(* IEC 61131-3 sources: MotionTestBenchMaster/Logical/00_AID/Libraries/Sidel_Libraries/Sidel_Obj, 21 files *)

(* ---- HMI_Structure.typ ---- *)
(*VALVES*)

TYPE
	HMI_Valve_Type : 	STRUCT  (*Valves Structure: Digital*)
		Out : BOOL; (*State: Output*)
		Alarm : BOOL; (*State: Position Alarm *)
		Opened : BOOL; (*State: Feed-Back Opened*)
		Closed : BOOL; (*State: Feed-Back Closed*)
		ConfigPosition : BOOL; (*Configuration: Valve Feed-Back Position Present *)
		ConfigPresent : BOOL; (*Configuration: Device Present*)
		ManOff : BOOL; (*Command: Manual Closed*)
		ManOn : BOOL; (*Command: Manual Opened *)
		Mask : BOOL; (*Command: Position Alarm Mask*)
		ManEnable : BOOL; (*Command Enable: Manual Enabled*)
		MaskEnable : BOOL; (*Command Enable: Mask Enabled*)
	END_STRUCT;
	HMI_Valve_MixProof_Type : 	STRUCT  (*Valves Structure: Digital Mix Proof*)
		Out : BOOL; (*State: Output*)
		Alarm : BOOL; (*State: Position Alarm *)
		Opened : BOOL; (*State: Feed-Back Opened*)
		Closed : BOOL; (*State: Feed-Back Closed*)
		ConfigPosition : BOOL; (*Configuration: Valve Feed-Back Position Present *)
		ConfigPresent : BOOL; (*Configuration: Device Present*)
		ManOff : BOOL; (*Command: Manual Closed*)
		ManOn : BOOL; (*Command: Manual Opened *)
		Mask : BOOL; (*Command: Position Alarm Mask*)
		ManEnable : BOOL; (*Command Enable: Manual Enabled*)
		MaskEnable : BOOL; (*Command Enable: Mask Enabled*)
		H_Out : BOOL; (*High State: Output*)
		H_Alarm : BOOL; (*High State: Position Alarm *)
		H_Opened : BOOL; (*High State: Feed-Back Opened*)
		H_Closed : BOOL; (*High State: Feed-Back Closed*)
		H_ConfigPosition : BOOL; (*High Configuration: Valve Closed State Present *)
		H_ManOff : BOOL; (*High Command: Manual Closed*)
		H_ManOn : BOOL; (*High Command: Manual Opened *)
		H_Mask : BOOL; (*High Command: Position Alarm Mask*)
		H_ManEnable : BOOL; (*High Command Enable: Manual Enabled*)
		H_MaskEnable : BOOL; (*High Command Enable: Mask Enabled*)
		L_Out : BOOL; (*Low State: Output*)
		L_Alarm : BOOL; (*Low State: Position Alarm *)
		L_Opened : BOOL; (*Low State: Feed-Back Opened*)
		L_Closed : BOOL; (*Low State: Feed-Back Closed*)
		L_ConfigPosition : BOOL; (*Low Configuration: Valve Closed State Present *)
		L_ManOff : BOOL; (*Low Command: Manual Closed*)
		L_ManOn : BOOL; (*Low Command: Manual Opened *)
		L_Mask : BOOL; (*Low Command: Position Alarm Mask*)
		L_ManEnable : BOOL; (*Low Command Enable: Manual Enabled*)
		L_MaskEnable : BOOL; (*Low Command Enable: Mask Enabled*)
	END_STRUCT;
	HMI_Valve_Mod_Type : 	STRUCT  (*Valves Structure: Analogic*)
		Out : BOOL; (*State: Output*)
		Alarm : BOOL; (*State: Position Alarm *)
		Opened : BOOL; (*State: Feed-Back Opened*)
		Closed : BOOL; (*State: Feed-Back Closed*)
		ConfigSlew : BOOL; (*Configuration: Output Slew Present*)
		ConfigPosition : BOOL; (*Configuration: Valve Feed-Back Position Present *)
		ConfigPresent : BOOL; (*Configuration: Device Present*)
		ManOff : BOOL; (*Command: Manual Closed*)
		ManOn : BOOL; (*Command: Drive Manual OUT = OUT_Man*)
		Mask : BOOL; (*Command: Position Alarm Mask*)
		ManEnable : BOOL; (*Command Enable: Manual Enabled*)
		MaskEnable : BOOL; (*Command Enable: Mask Enabled*)
		OUT_CV : REAL; (*State: Actual OUTPUT Control Value (0.0-:-100.0)*)
		OUT_Man : REAL; (*Command: Manual OUTPUT Value (0.0-:-100.0)*)
		FBK : REAL; (*State: Feed-Back INPUT Value (0.0-:-100.0)*)
	END_STRUCT;
END_TYPE

(*MOTORS*)

TYPE
	HMI_SCU_Type : 	STRUCT
		Visibility : BOOL;
		Alarm : BOOL;
		ErrCode : DINT;
		HwCmdUp : BOOL;
		HwCmdDown : BOOL;
		HwCmdStorePosition : BOOL;
	END_STRUCT;
	HMI_Column_Type : 	STRUCT
		Visibility : BOOL;
		Running : BOOL; (*State: Output*)
		Current : REAL;
		Initialized : BOOL;
		Position : REAL;
		Alarm : BOOL;
	END_STRUCT;
	HMI_Motor_Type : 	STRUCT  (*Motor Structure: Direct On Line*)
		Out : BOOL; (*State: Running*)
		Alarm : BOOL; (*State: Alarm (Isolated, Overload, FBK Fault)*)
		Isolated : BOOL; (*State: Motor Isolated*)
		Overload : BOOL; (*State: Overload*)
		FeedBack : BOOL; (*State: Feed-Back Fault*)
		ConfigPresent : BOOL; (*Configuration: Device Present*)
		ManOff : BOOL; (*Command: Manual Stop*)
		ManOn : BOOL; (*Command: Manual Start*)
		Mask : BOOL; (*Command: Alarm Mask*)
		ManEnable : BOOL; (*Command Enable: Manual Enabled*)
		MaskEnable : BOOL; (*Command Enable: Mask Enabled*)
	END_STRUCT;
	HMI_Motor_FC_Type : 	STRUCT  (*Motor Structure: Variable Frequency Drive*)
		Out : BOOL; (*State: Running *)
		Alarm : BOOL; (*State: Alarm (Isolated, Overload, FBK Fault)*)
		Isolated : BOOL; (*State: Motor Isolated*)
		Overload : BOOL; (*State: Overload*)
		FeedBack : BOOL; (*State: In Operation/Safe-OFF Feed-Back Fault*)
		BusFault : BOOL; (*State: Bus Control Fault*)
		Fault : BOOL; (*State: Inverter Internal Fault*)
		ConfigPresent : BOOL; (*Configuration: Device Present*)
		ManOff : BOOL; (*Command: Manual Stop*)
		ManOn : BOOL; (*Command: Manual Start*)
		Mask : BOOL; (*Command: Alarm Mask*)
		ManEnable : BOOL; (*Command Enable: Manual Enabled*)
		MaskEnable : BOOL; (*Command Enable: Mask Enabled*)
		OUT_CV : REAL; (*State: Actual OUTPUT Value (0.0-:-100.0)*)
		OUT_Man : REAL; (*Command: Manual OUTPUT Value (0.0-:-100.0)*)
	END_STRUCT;
	HMI_Dosing_Pump_Type : 	STRUCT  (*Motor Structure: Dosing Pump*)
		Out : BOOL; (*State: Running *)
		Alarm : BOOL; (*State: Alarm (Isolated, Overload, FBK Fault)*)
		Isolated : BOOL; (*State: Motor Isolated*)
		Overload : BOOL; (*State: Overload*)
		FeedBack : BOOL; (*State: In Operation/Safe-OFF Feed-Back Fault*)
		Pulse_FBK : BOOL; (*State: Pulse Feed-Back Alarm*)
		Internal_Fault : BOOL; (*State: Internal Alarm*)
		ConfigPresent : BOOL; (*Configuration: Device Present*)
		ManOff : BOOL; (*Command: Manual Stop*)
		ManOn : BOOL; (*Command: Manual Start *)
		Mask : BOOL; (*Command: Alarm Mask*)
		ManEnable : BOOL; (*Command Enable: Manual Enabled*)
		MaskEnable : BOOL; (*Command Enable: Mask Enabled*)
		Stroke_Value : REAL; (*Setting CC/Stroke [cm3/stroke]*)
		Concentration : REAL; (*Tank Concentrated percentage [0..1000000 ppm]*)
		Density : REAL; (*Specific Weight [kg]*)
	END_STRUCT;
	HMI_Danfoss_Diag_Type : 	STRUCT
		PCV : HMI_Danfoss_PCV_Type;
		PCD_Read : HMI_Danfoss_PCD_Read_Type;
	END_STRUCT;
	HMI_Danfoss_PCV_Type : 	STRUCT
		Alarm : DINT;
	END_STRUCT;
	HMI_Danfoss_PCD_Read_Type : 	STRUCT
		Power : REAL;
		Motor_Current : REAL;
		Frequency : REAL;
		Torque : REAL;
		Main_Actual_Value : REAL;
		Speed_RPM : REAL;
		Status_Word : UINT;
	END_STRUCT;
	HMI_Fan_Type : 	STRUCT
		HMI_Pressurizer : ARRAY[1..6]OF HMI_Pressurizer_Type; (*Single Fans to HMI*)
		HMI_Galvani : HMI_Galvani_Type; (*Galvani Roof Fans*)
	END_STRUCT;
	HMI_Galvani_Type : 	STRUCT
		Out : BOOL;
		ConfigPresent : BOOL; (*Configuration: Device Present*)
		SS2P_Lamp1 : HMI_SS2P_Type; (*SS2P Lamp*)
		SS2P_Lamp2 : HMI_SS2P_Type; (*SS2P Lamp*)
		ManState : BOOL; (*State: Device in manual mode*)
		ManEnable : BOOL; (*Command Enable: Manual Enabled*)
		ManFlowSet : BOOL; (*Command: Manual Flow set command*)
		ManOff : BOOL; (*Command: Manual Stop*)
		ManOn : BOOL; (*Command: Manual Start*)
		MaskEnable : BOOL; (*Command Enable: Mask Enabled*)
		Mask : BOOL; (*Command: Alarm Mask*)
		FlowSet : BOOL; (*State: Flow set speed *)
		Alarm : BOOL; (*State: Alarm (Isolated, Overload, FBK Fault)*)
		AlarmAbsoluteFilter : BOOL; (*Fault : Absolute filter clogged*)
		AlarmPrefilterExt : BOOL; (*Fault : External PreFilter Clogged*)
		AlarmPrefilterInt : BOOL; (*Fault : Internal PreFilter Clogged*)
		Overload : BOOL; (*State: Power supply on*)
	END_STRUCT;
	HMI_Pressurizer_Type : 	STRUCT
		Out : BOOL;
		ConfigPresent : BOOL; (*Configuration: Device Present*)
		SS2P_Lamp : HMI_SS2P_Type; (*SS2P Lamp*)
		ManState : BOOL; (*State: Device in manual mode*)
		ManEnable : BOOL; (*Command Enable: Manual Enabled*)
		ManOff : BOOL; (*Command: Manual Stop*)
		ManOn : BOOL; (*Command: Manual Start*)
		MaskEnable : BOOL; (*Command Enable: Mask Enabled*)
		Mask : BOOL; (*Command: Alarm Mask*)
		OUT_Man : REAL; (*Command :  Manual Speed OUT value selected (0 - 100)*)
		OUT_CV : REAL; (*State : Actual Speed OUT value %*)
		Alarm : BOOL; (*State: Alarm (Isolated, Overload, FBK Fault)*)
		AlarmFilter : BOOL; (*Fault : Absolute filter or PreFilter Clogged*)
	END_STRUCT;
	HMI_GreasingPump_Type : 	STRUCT
		LowLevel : HMI_DI_Type;
		CycleEnd : HMI_DI_Type;
		Motor : HMI_Motor_Type;
	END_STRUCT;
END_TYPE

(*INSTRUMENTS*)

TYPE
	HMI_Valve_Ejector_Type : 	STRUCT  (*Valves Structure: Digital*)
		Out : BOOL; (*State: Output*)
		Alarm : BOOL; (*State: Position Alarm *)
		Opened : BOOL; (*State: Feed-Back Opened*)
		Closed : BOOL; (*State: Feed-Back Closed*)
		ConfigPosition : BOOL; (*Configuration: Valve Feed-Back Position Present *)
		ConfigPresent : BOOL; (*Configuration: Device Present*)
		ManOff : BOOL; (*Command: Manual Closed*)
		ManOn : BOOL; (*Command: Manual Opened *)
		Mask : BOOL; (*Command: Position Alarm Mask*)
		ManEnable : BOOL; (*Command Enable: Manual Enabled*)
		MaskEnable : BOOL; (*Command Enable: Mask Enabled*)
		CounterReset : BOOL; (*Command: Reset Counter*)
		TotalErrors : UDINT; (*State : Total Errors*)
		AbsoluteErrors : USINT; (*State : Absolute Errors*)
		ConsecutiveErrors : USINT; (*State : Consecutive Errors*)
	END_STRUCT;
	HMI_Photocell_Type : 	STRUCT  (*Instrument Structure: Photocell*)
		On : BOOL; (*State: Active*)
		Alarm : BOOL; (*State: Alarm*)
		Wait : BOOL; (*State: Waiting condition*)
		ConfigAlarm : BOOL; (*Configuration: Alarm Present*)
		ConfigPresent : BOOL; (*Configuration: Instrument Present*)
		Mask : BOOL; (*Command: Alarm Mask*)
		MaskEnable : BOOL; (*Command Enable: Mask Enabled*)
		CounterReset : BOOL; (*Command: Reset Counter*)
		TotalErrors : UDINT; (*State : Total Errors*)
		RepetitiveErrors : USINT; (*State : Repetitive Errors*)
		AbsoluteErrors : USINT; (*State : Absolute Errors*)
		ConsecutiveErrors : USINT; (*State : Consecutive Errors*)
		AlwaysTrueSteps : USINT;
	END_STRUCT;
	HMI_DI_Type : 	STRUCT  (*Instrument Structure: Digital*)
		On : BOOL; (*State: Active*)
		Alarm : BOOL; (*State: Alarm*)
		Wait : BOOL; (*State: Waiting condition*)
		ConfigAlarm : BOOL; (*Configuration: Alarm Present*)
		ConfigPresent : BOOL; (*Configuration: Instrument Present*)
		Mask : BOOL; (*Command: Alarm Mask*)
		MaskEnable : BOOL; (*Command Enable: Mask Enabled*)
	END_STRUCT;
	HMI_Analog_IN_Type : 	STRUCT  (*Instrument Structure: Analogic*)
		Alarm : BOOL; (*State: Instrument in fault (Probe Fault)*)
		Wait : BOOL; (*State: Waiting condition*)
		WaitCounter : BOOL; (*State: Waiting Counter condition*)
		ConfigPopUp : BOOL; (*Configuration: Instrument Pop-Up Present (TRUE=Pop-Up NOT Present)*)
		ConfigTot : BOOL; (*Configuration: Totalizator Present (TRUE=Totalizator Present)*)
		ConfigAlarm : BOOL; (*Configuration: Alarm Present (TRUE=Command Mask Present)*)
		ConfigPresent : BOOL; (*Configuration: Instrument Present*)
		ConfigCounter : BOOL; (*Configuration: Counter Present*)
		ResetTot : BOOL; (*Command: Totalizator Reset*)
		Mask : BOOL; (*Command: Alarm Mask (Probe Fault disabled)*)
		MaskEnable : BOOL; (*Command Enable: Mask Enabled*)
		PV : REAL; (*Input: Scaled Process Value*)
		SP : REAL; (*Input: Actual SetPoint*)
		PV_Counter : REAL; (*Input: Counter Current Value*)
		SP_Counter : REAL; (*Input: Counter Requested Value*)
		Tot : REAL; (*Input: Totalizator*)
	END_STRUCT;
	HMI_Analog_IN_Mode_Type : 	STRUCT  (*Instrument Structure: Analogic Multi Scale*)
		Mode : ARRAY[0..3]OF HMI_Analog_IN_Type;
	END_STRUCT;
	HMI_Analog_Multiscale_Type : 	STRUCT  (*Instrument Structure: Analogic*)
		Alarm : BOOL; (*State: Instrument in fault (Probe Fault)*)
		Unit : USINT; (*0 = Unit1 ; 1 = Unit2 ; 2 = Unit3 ; etc...*)
		ConfigPopup : BOOL; (*Configuration: Instrument Pop-Up Present (TRUE=Pop-Up NOT Present)*)
		ConfigAlarm : BOOL; (*Configuration: Alarm Present (TRUE=Command Mask Present)*)
		ConfigPresent : BOOL; (*Configuration: Instrument Present*)
		ResetTot : BOOL; (*Command: Totalizator Reset*)
		Mask : BOOL; (*Command: Alarm Mask (Probe Fault disabled)*)
		MaskEnable : BOOL; (*Command Enable: Mask Enabled*)
		Wait : ARRAY[0..3]OF BOOL; (*State: Waiting condition*)
		ConfigTot : ARRAY[0..3]OF BOOL; (*Configuration: Totalizator Present (TRUE=Totalizator Present)*)
		WaitCounter : ARRAY[0..3]OF BOOL; (*State: Waiting Counter condition*)
		ConfigCounter : ARRAY[0..3]OF BOOL; (*Configuration: Counter Present*)
		PV : ARRAY[0..3]OF REAL; (*Input: Scaled Process Value*)
		SP : ARRAY[0..3]OF REAL; (*Input: Actual SetPoint*)
		PV_Counter : ARRAY[0..3]OF REAL; (*Input: Counter Current Value*)
		SP_Counter : ARRAY[0..3]OF REAL; (*Input: Counter Requested Value*)
		Tot : ARRAY[0..3]OF REAL; (*Input: Totalizator*)
	END_STRUCT;
	HMI_TNK_Level_Type : 	STRUCT
		CFG_Level_Percentage : BOOL;
		Level_Percentage : REAL; (*[%]*)
		CFG_Level_Percentage_SP : BOOL; (*[%]*)
		Level_Height_SP : REAL; (*[mm]*)
		Level_Percentage_SP : REAL; (*[%]*)
		CFG_Volume : BOOL;
		Volume : REAL; (*[l]*)
		CFG_Volume_SP : BOOL; (*[l]*)
		Level_Percentage_Wait : BOOL;
		Level_Height_Wait : BOOL;
		Volume_Wait : BOOL;
		Volume_SP : REAL; (*[l]*)
		CFG_Level_Height : BOOL;
		Level_Height : REAL; (*[mm]*)
	END_STRUCT;
	HMI_TNK_Level_v00_Type : 	STRUCT
		ConfigPresent : BOOL := TRUE;
		TNK_Height_mm : REAL; (*[mm]*)
		TNK_Height_Sp : REAL; (*[mm]*)
		TNK_Height_Wait : BOOL;
		TNK_Percentage : REAL; (*[%]*)
		TNK_Percentage_Sp : REAL; (*[%]*)
		TNK_Percentage_Wait : BOOL;
		TNK_Volume_liters : REAL; (*[l]*)
		TNK_Volume_Sp : REAL; (*[l]*)
		TNK_Volume_Wait : BOOL;
	END_STRUCT;
	HMI_GateDoor_Type : 	STRUCT
		Opened : BOOL;
		ShortSafety : BOOL;
		Production : HMI_DI_Type;
		Cleaning : HMI_DI_Type;
	END_STRUCT;
END_TYPE

(*PID*)

TYPE
	HMI_PID_Mode_Type : 	STRUCT
		Mode : ARRAY[0..3]OF HMI_PID_Type;
	END_STRUCT;
	HMI_PID_Type : 	STRUCT  (*PID Structure: PID Control*)
		Enable : BOOL; (*State: PID Enable*)
		Mode : BOOL; (*State: PID Mode (Automatic = 1  Manual = 0)*)
		Alarm : BOOL; (*State: PID PV in fault*)
		SP_Obtained : BOOL; (*State: PID Set Point Reached*)
		SP_SlewRunning : BOOL; (*State: PID Set Point Slew Running*)
		CnScale : BOOL; (*Configuration: FF and PID OUT Scale - TRUE-> 0-100%, FALSE-> Ing.Unit.*)
		ConfigSlewPresent : BOOL; (*Configuration: Slew Present*)
		ConfigPresent : BOOL; (*Configuration : PID present*)
		SPLocal : BOOL; (*Command: PID Manual Set Point -> "SP_Local"*)
		PV : REAL; (*State: PID Process Value*)
		SP_Actual : REAL; (*State: PID Set Point in Use*)
		SP_Target : REAL; (*State: PID Set Point*)
		FF_OUT : REAL; (*State: PID Feed Forward calculated value*)
		OUT : REAL; (*State: PID Output*)
		SP_Local : REAL; (*Command: PID Manual Set Point Target Value*)
	END_STRUCT;
END_TYPE

(*PWM*)

TYPE
	HMI_PWM_Type : 	STRUCT  (*PWM Structure: Pulse Width Modulation*)
		Out : BOOL; (*State: On*)
		Alarm : BOOL; (*State: Alarm (Isolated, Overload, FBK Fault)*)
		Isolated : BOOL; (*State: Isolated*)
		Overload : BOOL; (*State: Overload*)
		FeedBack : BOOL; (*State: Feed-Back Fault*)
		ConfigPresent : BOOL; (*Configuration: Device Present*)
		ManOff : BOOL; (*Command: Manual Stop*)
		ManOn : BOOL; (*Command: Manual Start*)
		Mask : BOOL; (*Command: Alarm Mask*)
		ManEnable : BOOL; (*Command Enable: Manual Enabled*)
		MaskEnable : BOOL; (*Command Enable: Mask Enabled*)
		OUT_CV : REAL; (*State: Actual OUTPUT Control Value (0.0-:-100.0)*)
		OUT_Man : REAL; (*Command: Manual OUTPUT Value (0.0-:-100.0)*)
	END_STRUCT;
END_TYPE

(* *)

TYPE
	HMI_SS2P_Type : 	STRUCT  (*Selector 2 position (Auto-Man; ON-OFF;) 0=Auto/OFF - 1=Man/ON*)
		Enable : BOOL; (*State: Command Enabled*)
		LampON : BOOL; (*State: Lamp Command ON*)
		Blink : BOOL; (*State: Blink LampOn*)
		Visibility : BOOL; (*Configuration: Present*)
		ON : BOOL; (*Command: Selector Button ON*)
	END_STRUCT;
END_TYPE

(* ---- IO_Structure.typ ---- *)
(*VALVES*)

TYPE
	IO_Valve_Mod_Type : 	STRUCT
		AO_Raw : INT;
		AI_Raw : INT;
		Valve : IO_Valve_Type;
	END_STRUCT;
	IO_ValveMac_Type : 	STRUCT
		DI_PowerSupplyPhyChannelOk : BOOL;
		DI_Opened : BOOL; (*DI Valve Open - Feedback*)
		DI_Closed : BOOL; (*DI Valve Close - Feedback*)
		DO_Opened : BOOL; (*DO Valve Open*)
		DO_Closed : BOOL; (*DO Valve Close*)
	END_STRUCT;
	IO_Valve_Type : 	STRUCT
		DI_Opened : BOOL; (*DI Valve Open - Feedback*)
		DI_Closed : BOOL; (*DI Valve Close - Feedback*)
		DO_Opened : BOOL; (*DO Valve Open*)
		DO_Closed : BOOL; (*DO Valve Close*)
	END_STRUCT;
END_TYPE

(*MOTORS*)

TYPE
	IO_Motor_FwBw_Type : 	STRUCT  (*Motor control Forward Backward*)
		DI_SafetyEnable : BOOL; (*Safety Enable from IOMapping*)
		DI_SafetyFault : BOOL; (*Safety Feed-Back from Safety CPU*)
		DI_Fault : BOOL;
		DI_ContactorFBK : BOOL; (*Contactor Feed-Back *)
		DI_OverloadOK : BOOL := TRUE; (*Not present in case of UL*)
		DI_ManSwitchON : BOOL := TRUE;
		DO_MotorFw : BOOL; (*Start Forward*)
		DO_MotorBw : BOOL; (*Start Backward*)
	END_STRUCT;
	IO_MotorFC280_Type : 	STRUCT  (*Motor control*)
		DI_SafetyEnable : BOOL; (*Safety Enable from IOMapping*)
		DI_SafetyFault : BOOL; (*Safety Feed-Back from Safety CPU*)
		DI_ManSwitchON : BOOL := TRUE;
		DI_ContactorFBK : BOOL; (*Contactor Feed-Back *)
		DI_OverloadOK : BOOL := TRUE; (*Not present in case of UL*)
		DO_MotorON : BOOL; (*Start*)
		DO_ShuntTrip : BOOL; (*Thermal Protection Forced Trip*)
	END_STRUCT;
	IO_Motor_Type : 	STRUCT  (*Motor control*)
		DI_SafetyEnable : BOOL; (*Safety Enable from IOMapping*)
		DI_SafetyFault : BOOL; (*Safety Feed-Back from Safety CPU*)
		DI_ManSwitchON : BOOL := TRUE;
		DI_ContactorFBK : BOOL; (*Contactor Feed-Back *)
		DI_OverloadOK : BOOL := TRUE; (*Not present in case of UL*)
		DO_MotorON : BOOL; (*Start*)
		DO_ShuntTrip : BOOL; (*Thermal Protection Forced Trip*)
	END_STRUCT;
	IO_UVtronic_Type : 	STRUCT  (*Henovia UV control*)
		DI_SafetyEnable : BOOL; (*Safety Enable from IOMapping*)
		DI_Ready : BOOL;
		DI_Alarm : BOOL;
		DI_GeneralFault : BOOL;
		DI_ContactorFBK : BOOL; (*Contactor Feed-Back *)
		DI_OverloadOK : BOOL := TRUE; (*Not present in case of UL*)
		DO_MotorON : BOOL; (*Start*)
	END_STRUCT;
	IO_PLK_DanfossFC280_Drive_Type : 	STRUCT  (*Powerlink Danfoss VLT Interface*)
		Input : IO_PLK_DanfossFC280_IN;
		Output : IO_PLK_DanfossFC280_OUT;
	END_STRUCT;
	IO_PLK_Danfoss_Drive_Type : 	STRUCT  (*Powerlink Danfoss VLT Interface*)
		Input : IO_PLK_Danfoss_IN;
		Output : IO_PLK_Danfoss_OUT;
	END_STRUCT;
	IO_PLK_DanfossFC280_IN : 	STRUCT  (*Powerlink Danfoss VLT Inputs*)
		STW : UINT; (*Status Word*)
		MAV : INT; (*Main Actual Value*)
		ActFreq : UDINT; (*Actual Frequency [Hz]*)
		ActCurrent : UINT; (*Actual Current [A]*)
		Power : UDINT; (*Power [kW]*)
		Torque : DINT; (*Torque [Nm]*)
		SpeedRPM : DINT; (*Speed [RPM]*)
		STW_EX : UDINT; (*Extended Status Word 1*)
		ErrorCode : UDINT; (*Error Code 1*)
		DigitalInput : UINT; (*Digital Input V4.A.A.1.6.13*)
	END_STRUCT;
	IO_PLK_Danfoss_IN : 	STRUCT  (*Powerlink Danfoss VLT Inputs*)
		STW : UINT; (*Status Word*)
		MAV : INT; (*Main Actual Value*)
		ActFreq : UINT; (*Actual Frequency [Hz]*)
		ActCurrent : DINT; (*Actual Current [A]*)
		Power : DINT; (*Power [kW]*)
		Torque : INT; (*Torque [Nm]*)
		SpeedRPM : DINT; (*Speed [RPM]*)
		STW_EX : UDINT; (*Extended Status Word 1*)
		ErrorCode : UDINT; (*Error Code 1*)
		DigitalInput : UINT; (*Digital Input V4.A.A.1.6.13*)
	END_STRUCT;
	IO_PLK_DanfossFC280_OUT : 	STRUCT  (*Powerlink Danfoss VLT Outputs*)
		CTW : UINT; (*Control Word*)
		MRW : INT; (*Main Reference Value*)
	END_STRUCT;
	IO_PLK_Danfoss_OUT : 	STRUCT  (*Powerlink Danfoss VLT Outputs*)
		CTW : UINT; (*Control Word*)
		MRW : INT; (*Main Reference Value*)
	END_STRUCT;
	IO_FanMain_Type : 	STRUCT
		DI_OverloadOK : BOOL := TRUE;
		DO_ZoneLighting : BOOL; (*V4.A.A.1.7.0*)
		Pressurizer : ARRAY[1..6]OF IO_Pressurizer_Type;
		GalvaniRoof : IO_GalvaniRoof_Type;
	END_STRUCT;
	IO_PressurizerMain_Type : 	STRUCT
		DI_OverloadOK : BOOL := TRUE;
		Pressurizer : ARRAY[1..6]OF IO_Pressurizer_Type;
	END_STRUCT;
	IO_GalvaniRoof_Type : 	STRUCT
		DI_Running : BOOL;
		DI_AbsoluteFilterAlarm : BOOL;
		DI_PrefilterExtAlarm : BOOL;
		DI_PrefilterIntAlarm : BOOL;
		DI_CabinetPoweredOn : BOOL;
		DO_Start : BOOL;
		DO_FlowSet : BOOL;
		DO_LightingArea_1 : BOOL;
		DO_LightingArea_2 : BOOL;
	END_STRUCT;
	IO_Pressurizer_Type : 	STRUCT
		DO_Lighting : BOOL;
		AO_Raw : INT;
		DI_PressurizerON : BOOL; (*Pressurizzer ON*)
		DI_PrefilterAlarm : BOOL; (*Pressurizzer prefilter clogged*)
		DI_AbsoluteFilterAlarm : BOOL; (*Pressurizzer absolute filter clogged*)
	END_STRUCT;
	IO_MotionFan_Type : 	STRUCT
		DI_ManSwitchON : BOOL := TRUE;
		DI_OverloadOK : BOOL := TRUE;
		DI_ContactorFBK : BOOL := TRUE;
		DO_MotorON : BOOL;
	END_STRUCT;
END_TYPE

(*INSTRUMENTS*)

TYPE
	IO_Analog_IN_OUT_Type : 	STRUCT
		AO_Raw : INT := 0; (*Analog Input From HW*)
		AI : IO_Analog_IN_Type; (*Analog Input From HW*)
	END_STRUCT;
	IO_Analog_IN_Type : 	STRUCT
		AI_Raw : INT := 0; (*Analog Input From HW*)
		DI_ChannelOk : BOOL := TRUE;
		DI_Pulse : BOOL; (*Totalizer Pulse*)
		DI_Alarm : BOOL; (*Instrument Alarm*)
		DO_SetScale : BOOL; (*Scale Change Output*)
	END_STRUCT;
	IO_Digital_IN_Type : 	STRUCT
		DI_Input : BOOL;
	END_STRUCT;
	IO_Digital_OUT_Type : 	STRUCT
		DO_Output : BOOL;
	END_STRUCT;
	IO_GreasingPump_Type : 	STRUCT
		LowLevel : IO_Digital_IN_Type;
		CycleEnd : IO_Digital_IN_Type;
		Motor : IO_Motor_Type;
	END_STRUCT;
	IN_Analog_Multiscale : 	STRUCT
		ScaleLOW : REAL;
		ScaleHIGH : REAL;
		ActualSP : REAL; (*Signal Input Actual Set Point*)
		MinDev : REAL; (*To Set Point Low Deviation (for SP obtained)*)
		MaxDev : REAL; (*To Set Point High Deviation (for SP obtained)*)
		WaitDelay : TIME;
		HighLimitEn : BOOL;
		HighLimitSP : REAL;
		HighLimitHyst : REAL;
		HighLimitDelay : TIME;
		LowLimitEn : BOOL;
		LowLimitSP : REAL;
		LowLimitHyst : REAL;
		LowLimitDelay : TIME;
		TotPulseWeight : REAL;
		TotType : USINT;
		PLCCounterSP : REAL;
		PLCCounterReset : BOOL;
		HMITotEn : BOOL;
		HMITotReset : BOOL;
	END_STRUCT;
	OUT_Analog_Multiscale : 	STRUCT
		ActValue : REAL; (*Manipulated value*)
		LowLimit : BOOL;
		HighLimit : BOOL;
		PLCCounterReached : BOOL; (*Output Fault*)
		Active : BOOL; (*Request to Instrument Scale Activation*)
	END_STRUCT;
	IO_IncrementalEncoder : 	STRUCT  (*//V4.A.A.1.6.11*)
		CountAtZero : DINT;
		Counter : INT;
		Status : USINT;
		Reference : USINT;
		DI_EnableReference : IO_Digital_IN_Type;
		DI_NotPowered : IO_Digital_IN_Type;
	END_STRUCT;
END_TYPE

(* ---- Local_Structure.typ ---- *)
TYPE
	Danfoss_Event_Type : 	STRUCT
		Brake_Check : BOOL;
		Drive_Over_Temperature : BOOL;
		Earth_Fault : BOOL;
		Control_Card_Over_Temperature : BOOL;
		Controlword_timeout : BOOL;
		Over_Current : BOOL;
		Torque_Limit : BOOL;
		Motor_Thermistor_Over_Temp : BOOL;
		Motor_ETR_Over_Temperature : BOOL;
		Inverter_Over_Loaded : BOOL;
		DC_Link_Under_Voltage : BOOL;
		DC_Link_Over_Voltage : BOOL;
		Short_Circuit : BOOL;
		Inrush_Fault : BOOL;
		Mains_Phase_Loss : BOOL;
		AMA_not_OK : BOOL;
		Live_Zero_Error : BOOL;
		Internal_Fault : BOOL;
		Brake_Resistor_Power_Limit : BOOL;
		Motor_Phase_U_Missing : BOOL;
		Motor_Phase_V_Missing : BOOL;
		Motor_Phase_W_Missing : BOOL;
		Fieldbus_Communication_Fault : BOOL;
		_24V_Supply_Fault : BOOL;
		Mains_Faliure : BOOL;
		_2V_Supply_Fault : BOOL;
		Brake_Resistor_Short_Circuit : BOOL;
		Brake_Chopper_Fault : BOOL;
		Configuration_Option_Change : BOOL;
		Drive_Initialisation : BOOL;
		Safe_Stop : BOOL;
		Mecanical_Brake_Low : BOOL;
	END_STRUCT;
	Danfoss_STW_Type : 	STRUCT
		Speed_Referece : BOOL;
		Fault : BOOL;
		Warning : BOOL;
		In_Operation : BOOL;
		T37_Ready : BOOL;
	END_STRUCT;
	Danfoss_DI_Type : 	STRUCT  (*V4.A.A.1.6.13*)
		T33 : BOOL;
		T32 : BOOL;
		T29 : BOOL;
		T27 : BOOL;
		T19 : BOOL;
		T18 : BOOL;
		T37 : BOOL;
		Bit7 : BOOL;
		Bit8 : BOOL;
		Bit9 : BOOL;
		Bit10 : BOOL;
		Bit11 : BOOL;
		Bit12 : BOOL;
		Bit13 : BOOL;
		Bit14 : BOOL;
		Bit15 : BOOL;
	END_STRUCT;
	Danfoss_CTW_Type : 	STRUCT
		Coasting : BOOL;
		Hold_Output_Frequency : BOOL;
		DC_Brake : BOOL;
		Quick_Stop : BOOL;
		Start : BOOL;
		Reset : BOOL;
		Reverse : BOOL;
		Data_Valid : BOOL;
	END_STRUCT;
	FanZoneAlarm_Type : 	STRUCT
		PressurizerZone : PressurizerAlarm_Type;
		Pressurizer : ARRAY[1..6]OF PressurizerAlarm_Type;
		Galvani : GalvaniAlarm_Type;
	END_STRUCT;
	GalvaniAlarm_Type : 	STRUCT
		RunningAlarm : BOOL;
		AbsoluteFilterAlarm : BOOL;
		PrefilterExtAlarm : BOOL;
		PrefilterIntAlarm : BOOL;
		CabinetAlarm : BOOL;
		Overload : BOOL;
		SysSwitchedOff : BOOL;
		SysManSwitchedOff : BOOL;
	END_STRUCT;
	PressurizerZoneAlarm_Type : 	STRUCT
		PressurizerZone : PressurizerAlarm_Type;
		Pressurizer : ARRAY[1..6]OF PressurizerAlarm_Type;
	END_STRUCT;
	PressurizerAlarm_Type : 	STRUCT
		AbsoluteFilterAlarm : BOOL;
		PrefilterAlarm : BOOL;
		PressurizedOnAlarm : BOOL;
	END_STRUCT;
	ShiftPosition_Type : 	STRUCT
		ContainerPresence : BOOL;
		ContainerBlowedFault : BOOL;
		ContainerRinsed : BOOL;
		ContainerBurst : BOOL;
		ContainerFilled : BOOL;
		ContainerEjected : BOOL;
		ClosingReleased : BOOL;
		ContainerClosed : BOOL;
	END_STRUCT;
	ShiftPositionInfo :
		(
		ContainerPresence := 0,
		ContainerBlowedFault := 1,
		ContainerRinsed := 2,
		ContainerBurst := 3,
		ContainerFilled := 4,
		ContainerEjected := 5,
		ClosingReleased := 6,
		ContainerClosed := 7,
		EjectContainer := 8,
		ContainerPreClosed := 9, (*Master nuovo valore precedente 8*)
		DummyBottleInserted := 10,
		DummyContainerDisinserted := 11,
		ShiftPositionSpareBit12 := 12,
		ShiftPositionSpareBit13 := 13,
		ShiftPositionSpareBit14 := 14,
		ShiftPositionSpareBit15 := 15
		);
	BlowerInfo :
		(
		FillerContainerBlock := 0,
		ContainerBlowFault := 1,
		CombiContainerPresence := 2,
		BlowerInfoSpareBit03 := 3,
		BlowerInfoSpareBit04 := 4,
		BlowerInfoSpareBit05 := 5,
		BlowerInfoSpareBit06 := 6,
		BlowerInfoSpareBit07 := 7,
		BlowerInfoSpareBit08 := 8,
		BlowerInfoSpareBit09 := 9,
		BlowerInfoSpareBit10 := 10,
		BlowerInfoSpareBit11 := 11,
		BlowerInfoSpareBit12 := 12,
		BlowerInfoSpareBit13 := 13,
		BlowerInfoSpareBit14 := 14,
		BlowerInfoSpareBit15 := 15
		);
END_TYPE

(* ---- Analog_In.st ---- *)
FUNCTION_BLOCK Analog_In
	IF IN_ConfigPresent THEN

		(*****************************************************************)
		(****************************VALUE SCALING************************)
		(*****************************************************************)
		TON_ChannelOk(IN := IO.DI_ChannelOk, PT := t#400ms);

		IF IN_EngScale THEN
			VAR_ChannelActive := IO.AI_Raw < 32767;
		ELSIF TON_ChannelOk.Q THEN
			IF IN_0_20mA THEN
				VAR_ChannelActive := (IO.AI_Raw > 6000);
			ELSE
				VAR_ChannelActive := NOT ((IO.AI_Raw < -90) OR (IO.AI_Raw > 32767));
			END_IF
			OUT_RawOverflow 	:= (IO.AI_Raw > 32767) AND NOT HMI.Mask;
			OUT_RawUnderflow	:= NOT VAR_ChannelActive AND (IO.AI_Raw < 32767) AND NOT HMI.Mask;
		ELSE
			VAR_ChannelActive := FALSE;
			OUT_RawOverflow	  := FALSE;
			OUT_RawUnderflow  := FALSE;
		END_IF

		IF VAR_ChannelActive THEN
			IF IN_EngScale THEN
				VAR_Out := INT_TO_REAL(IO.AI_Raw) / 10.0;
			ELSE
				IF IN_0_20mA THEN
					LCRLimScal_0_20mA(
					x	:= INT_TO_REAL(IO.AI_Raw),
					x1	:= 6553.4,
					y1	:= IN_ScaleLOW,
					x2	:= 32767.0,
					y2	:= IN_ScaleHIGH
					);

					VAR_Out := LCRLimScal_0_20mA.y;
				ELSE
					LCRLimScal_4_20mA(
					x	:= INT_TO_REAL(IO.AI_Raw),
					x1	:= 0.0,
					y1	:= IN_ScaleLOW,
					x2	:= 32767.0,
					y2	:= IN_ScaleHIGH
					);

					VAR_Out := LCRLimScal_4_20mA.y;
				END_IF
			END_IF
		END_IF

		(*****************************************************************)
		(****************************FAULTS*******************************)
		(*****************************************************************)
		IF OUT_RawOverflow OR OUT_RawUnderflow THEN
			VAR_iFault := NOT VAR_Mask;
		ELSIF IN_Reset THEN
			VAR_iFault	:= FALSE;
		END_IF

		IF NOT IN_Simulation THEN
			OUT_ActValue 	:= VAR_Out;
			VAR_Mask		:= HMI.Mask AND IN_MaskEn;
			VAR_Fault 		:= VAR_iFault;
		ELSE
			OUT_ActValue 	:= HMI.PV;
			VAR_Mask		:= HMI.Mask;
			VAR_Fault 		:= FALSE;
		END_IF

		IF VAR_Fault THEN
			IF IN_FaultOutMode = CST_AI_FaultMode_Low THEN
				VAR_Out := IN_ScaleLOW;
			ELSIF IN_FaultOutMode = CST_AI_FaultMode_High THEN
				VAR_Out := IN_ScaleHIGH;
			END_IF
			OUT_Alarm := NOT VAR_Mask;
		ELSIF IN_Reset THEN
			OUT_Alarm := FALSE;
		END_IF

		(*****************************************************************)
		(****************************LIMITS*******************************)
		(*****************************************************************)
		IF IN_HighLimitEn AND NOT VAR_Mask THEN
			TMR_TON_HighLimitDelay.IN := (OUT_ActValue >= IN_HighLimitSP);
			IF TMR_TON_HighLimitDelay.Q THEN
				OUT_HighLimit 	:= TRUE;
			ELSIF (OUT_ActValue <= (IN_HighLimitSP - IN_HighLimitHyst)) THEN
				OUT_HighLimit 	:= FALSE;
			END_IF
		ELSE
			TMR_TON_HighLimitDelay.IN 	:= FALSE;
			OUT_HighLimit 				:= FALSE;
		END_IF
		TMR_TON_HighLimitDelay(PT := IN_HighLimitDelay);

		IF IN_LowLimitEn AND NOT VAR_Mask THEN
			TMR_TON_LowLimitDelay.IN := (OUT_ActValue <= IN_LowLimitSP);
			IF TMR_TON_LowLimitDelay.Q THEN
				OUT_LowLimit 	:= TRUE;
			ELSIF (OUT_ActValue >= (IN_LowLimitSP + IN_LowLimitHyst)) THEN
				OUT_LowLimit 	:= FALSE;
			END_IF
		ELSE
			TMR_TON_LowLimitDelay.IN 	:= FALSE;
			OUT_LowLimit 				:= FALSE;
		END_IF
		TMR_TON_LowLimitDelay(PT := IN_LowLimitDelay);
		(*****************************************************************)
		(*************************COMPARE MODE****************************)
		(*****************************************************************)
		IF VAR_Mask THEN
			VAR_SpReached	:= TRUE;
			VAR_Wait		:= FALSE;
		ELSE
			CASE IN_CompareMode OF
				CST_AI_Compare_OFF:
					VAR_SpReached	:= FALSE;
					VAR_Wait		:= FALSE;
					HMI.SP			:= HMI.PV;

				CST_AI_Compare_LT:
					VAR_SpReached	:=  OUT_ActValue < (IN_ActualSP + IN_MinDev);
					VAR_Wait		:= NOT VAR_SpReached AND IN_AlarmEn;
					HMI.SP			:= IN_ActualSP;

				CST_AI_Compare_GT:
					VAR_SpReached	:=  OUT_ActValue > (IN_ActualSP - IN_MaxDev);
					VAR_Wait		:= NOT VAR_SpReached AND IN_AlarmEn;
					HMI.SP			:= IN_ActualSP;

				CST_AI_Compare_EQ:
					VAR_SpReached	:= (OUT_ActValue < (IN_ActualSP + IN_MaxDev)) AND (OUT_ActValue > (IN_ActualSP - IN_MinDev));
					VAR_Wait		:= NOT VAR_SpReached AND IN_AlarmEn;
					HMI.SP			:= IN_ActualSP;

				CST_AI_Compare_ON:
					VAR_SpReached	:= TRUE;
					VAR_Wait		:= FALSE;
					HMI.SP			:= HMI.PV;
			END_CASE
		END_IF
	ELSE
		VAR_SpReached 	:= TRUE;
		VAR_Wait		:= FALSE;
		HMI.SP			:= HMI.PV;
		OUT_LowLimit	:= FALSE;
		OUT_HighLimit 	:= FALSE;
	END_IF

	TMR_TOF_SpReached(IN:= VAR_SpReached, PT:= IN_WaitDelay);
	OUT_SpReached	:= TMR_TOF_SpReached.Q AND TON_ChannelOk.Q;

	(*****************************************************************)
	(***************************TOTALIZER*****************************)
	(*****************************************************************)
	IF IN_HMITotEn THEN
		HMITotalizer(
		IN_Pulse			:= IO.DI_Pulse,
		IN_AnalogPV			:= VAR_Out,
		IN_PulseWeight		:= IN_TotPulseWeight,
		IN_ConfigType		:= IN_TotType,
		IN_Reset			:= IN_HMITotReset OR HMI.ResetTot,
		OUT_TotalCounter	:= HMI.Tot);

		HMI.ConfigTot	:= TRUE;
	ELSE
		HMI.ConfigTot	:= FALSE;
		HMI.Tot 		:= 0.0;
	END_IF

	IF IN_PLCCounterEn THEN
		PLCCounter(
		IN_Pulse			:= IO.DI_Pulse,
		IN_AnalogPV			:= VAR_Out,
		IN_PulseWeight		:= IN_TotPulseWeight,
		IN_ConfigType		:= IN_TotType,
		IN_Reset			:= IN_PLCCounterReset,
		OUT_TotalCounter	:= HMI.PV_Counter);

		HMI.ConfigCounter	:= TRUE;
	ELSE
		HMI.ConfigCounter	:= FALSE;
		HMI.PV_Counter		:= 0.0;
	END_IF

	OUT_PLCCounterReached := (HMI.PV_Counter >= IN_PLCCounterSP);

	HMI.ConfigAlarm		:= IN_ConfigPopup;
	HMI.ConfigPresent 	:= IN_ConfigPresent;
	HMI.SP_Counter		:= IN_PLCCounterSP;
	HMI.WaitCounter		:= IN_PLCCounterEn AND NOT OUT_PLCCounterReached;
	HMI.Wait			:= VAR_Wait;
	HMI.Alarm			:= OUT_Alarm;
	HMI.PV 				:= OUT_ActValue;

	IF NOT IN_Simulation THEN
		HMI.MaskEnable	:= IN_MaskEn;
		HMI.ConfigPopUp	:= IN_ConfigPopup;
	ELSE
		HMI.MaskEnable	:= TRUE;
		HMI.ConfigPopUp	:= TRUE;
	END_IF
END_FUNCTION_BLOCK

(* ---- Analog_In_Direct_Inverse.st ---- *)
FUNCTION_BLOCK Analog_In_Direct_Inverse
	IF IN_ConfigPresent THEN

		(*****************************************************************)
		(****************************VALUE SCALING************************)
		(*****************************************************************)
		IF IN_EngScale THEN
			VAR_ChannelActive := IO.AI_Raw < 32767;
		ELSE
			IF IN_0_20mA THEN
				VAR_ChannelActive := (IO.AI_Raw > 6000);
			ELSE
				VAR_ChannelActive := NOT ((IO.AI_Raw < -90) OR (IO.AI_Raw > 32767));
			END_IF
			OUT_RawOverflow 	:= (IO.AI_Raw > 32767) AND NOT HMI.Mask;
			OUT_RawUnderflow	:= NOT VAR_ChannelActive AND (IO.AI_Raw < 32767) AND NOT HMI.Mask;
		END_IF

		LCRLimScal_0_20mA(
		x	:= INT_TO_REAL(IO.AI_Raw),
		x1	:= 6553.4,
		y1	:= IN_ScaleLOW,
		x2	:= 32767.0,
		y2	:= IN_ScaleHIGH
		);

		LCRLimScal_4_20mA(
		x	:= INT_TO_REAL(IO.AI_Raw),
		x1	:= 0.0,
		y1	:= IN_ScaleLOW,
		x2	:= 32767.0,
		y2	:= IN_ScaleHIGH
		);

		IF VAR_ChannelActive THEN
			IF IN_EngScale THEN
				VAR_Out := INT_TO_REAL(IO.AI_Raw) / 10.0;
			ELSE
			    IF IN_0_20mA AND IN_Direct_Inverse THEN
					VAR_Out := IN_Delta + (IN_ScaleHIGH - IN_ScaleLOW) - LCRLimScal_0_20mA.y;
				ELSIF NOT IN_0_20mA AND IN_Direct_Inverse THEN
					VAR_Out := IN_Delta + (IN_ScaleHIGH - IN_ScaleLOW) - LCRLimScal_4_20mA.y;
				ELSIF IN_0_20mA AND NOT IN_Direct_Inverse THEN
					VAR_Out := IN_Delta + LCRLimScal_0_20mA.y;
				ELSIF NOT IN_0_20mA AND NOT IN_Direct_Inverse THEN
					VAR_Out := IN_Delta + LCRLimScal_4_20mA.y;
				END_IF
			END_IF

			IF IN_Reset THEN
				VAR_iFault := FALSE;
			END_IF
		ELSE
			VAR_iFault := NOT VAR_Mask;
		END_IF

		(*****************************************************************)
		(***********************FAULTS AND LIMITS*************************)
		(*****************************************************************)
		IF NOT IN_Simulation THEN
			OUT_ActValue 	:= VAR_Out;
			VAR_Mask		:= HMI.Mask AND IN_MaskEn AND IN_AlarmEn ;
			VAR_Fault 		:= VAR_iFault;
		ELSE
			OUT_ActValue 	:= HMI.PV;
			VAR_Mask		:= HMI.Mask;
			VAR_Fault 		:= FALSE;
		END_IF

		IF VAR_Fault AND IN_AlarmEn THEN
			IF IN_FaultOutMode = CST_AI_FaultMode_Low THEN
				VAR_Out := IN_ScaleLOW;
			ELSIF IN_FaultOutMode = CST_AI_FaultMode_High THEN
				VAR_Out := IN_ScaleHIGH;
			END_IF
			OUT_Alarm := TRUE;
		ELSIF IN_Reset THEN
			OUT_Alarm := FALSE;
		END_IF

		IF IN_HighLimitEn AND NOT VAR_Mask THEN
			TMR_TON_HighLimitDelay(	IN := (OUT_ActValue >= IN_HighLimitSP),
			PT := IN_HighLimitDelay);

			IF TMR_TON_HighLimitDelay.Q THEN
				OUT_HighLimit 	:= TRUE;
			ELSIF (OUT_ActValue <= (IN_HighLimitSP - IN_HighLimitHyst)) THEN
				OUT_HighLimit 	:= FALSE;
			END_IF
		ELSE
			OUT_HighLimit := FALSE;
		END_IF

		IF IN_LowLimitEn AND NOT VAR_Mask THEN
			TMR_TON_LowLimitDelay(	IN := (OUT_ActValue <= IN_LowLimitSP),
			PT := IN_LowLimitDelay);

			IF TMR_TON_LowLimitDelay.Q THEN
				OUT_LowLimit 	:= TRUE;
			ELSIF (OUT_ActValue >= (IN_LowLimitSP + IN_LowLimitHyst)) THEN
				OUT_LowLimit 	:= FALSE;
			END_IF
		ELSE
			OUT_LowLimit := FALSE;
		END_IF

		(*****************************************************************)
		(*************************COMPARE MODE****************************)
		(*****************************************************************)
		IF VAR_Mask THEN
			VAR_SpReached := TRUE;
			VAR_Wait := FALSE;
		ELSE
			CASE IN_CompareMode OF
				CST_AI_Compare_OFF:
					VAR_SpReached := FALSE;
					VAR_Wait := FALSE;
					HMI.SP	:= HMI.PV;

				CST_AI_Compare_LT:
					VAR_SpReached :=  OUT_ActValue < (IN_ActualSP + IN_MinDev);
					VAR_Wait := NOT VAR_SpReached;
					HMI.SP	:= IN_ActualSP;

				CST_AI_Compare_GT:
					VAR_SpReached :=  OUT_ActValue > (IN_ActualSP - IN_MaxDev);
					VAR_Wait := NOT VAR_SpReached;
					HMI.SP	:= IN_ActualSP;

				CST_AI_Compare_EQ:
					VAR_SpReached := (OUT_ActValue < (IN_ActualSP + IN_MaxDev)) AND (OUT_ActValue > (IN_ActualSP - IN_MinDev));
					VAR_Wait := NOT VAR_SpReached;
					HMI.SP	:= IN_ActualSP;

				CST_AI_Compare_ON:
					VAR_SpReached := TRUE;
					VAR_Wait := FALSE;
					HMI.SP	:= HMI.PV;
			END_CASE
		END_IF
	ELSE
		OUT_SpReached 			:= TRUE;
		OUT_LowLimit			:= FALSE;
		OUT_HighLimit 			:= FALSE;
	END_IF

	TMR_TOF_SpReached(IN:= VAR_SpReached, PT:= IN_WaitDelay);
	OUT_SpReached	:= TMR_TOF_SpReached.Q;

	HMI.ConfigAlarm		:= IN_AlarmEn;
	HMI.ConfigPresent 	:= IN_ConfigPresent;
	HMI.Wait			:= VAR_Wait;
	HMI.Alarm			:= OUT_Alarm;
	HMI.PV 				:= OUT_ActValue;

	IF NOT IN_Simulation THEN
		HMI.MaskEnable	:= IN_MaskEn;
		HMI.ConfigPopUp	:= IN_ConfigPopup;
	ELSE
		HMI.MaskEnable	:= TRUE;
		HMI.ConfigPopUp	:= TRUE;
	END_IF

END_FUNCTION_BLOCK

(* ---- Analog_In_Multicompare.st ---- *)
FUNCTION_BLOCK Analog_In_Multicompare
	IF IN_ConfigPresent THEN

	(*****************************************************************)
	(****************************VALUE SCALING************************)
	(*****************************************************************)
		IF IN_EngScale THEN
			VAR_ChannelActive := IO.AI_Raw < 32767;
		ELSE
			IF IN_0_20mA THEN
				VAR_ChannelActive := (IO.AI_Raw > 6000);
			ELSE
				VAR_ChannelActive := NOT ((IO.AI_Raw < -90) OR (IO.AI_Raw > 32767));
			END_IF
			OUT_RawOverflow 	:= (IO.AI_Raw > 32767) AND NOT HMI.Mask;
			OUT_RawUnderflow	:= NOT VAR_ChannelActive AND (IO.AI_Raw < 32767) AND NOT HMI.Mask;
		END_IF

		VAR_Index := IN_ScaleIndex;

		LCRLimScal_0_20mA(
			x	:= INT_TO_REAL(IO.AI_Raw),
			x1	:= 6553.4,
			y1	:= IN_Scale[VAR_Index].ScaleLOW,
			x2	:= 32767.0,
			y2	:= IN_Scale[VAR_Index].ScaleHIGH
			);

		LCRLimScal_4_20mA(
			x	:= INT_TO_REAL(IO.AI_Raw),
			x1	:= 0.0,
			y1	:= IN_Scale[VAR_Index].ScaleLOW,
			x2	:= 32767.0,
			y2	:= IN_Scale[VAR_Index].ScaleHIGH
			);

		IF VAR_ChannelActive THEN
			IF IN_EngScale THEN
				VAR_Out := INT_TO_REAL(IO.AI_Raw) / 10.0;
			ELSE
				IF IN_0_20mA THEN
					VAR_Out := LCRLimScal_0_20mA.y;
				ELSE
					VAR_Out := LCRLimScal_4_20mA.y;
				END_IF
			END_IF

			IF IN_Reset THEN
				VAR_iFault := FALSE;
			END_IF
		ELSE
			VAR_iFault := NOT VAR_Mask;
		END_IF

	(*****************************************************************)
	(***********************FAULTS AND LIMITS*************************)
	(*****************************************************************)
		IF NOT IN_Simulation THEN
			OUT_Scale[VAR_Index].ActValue 	:= VAR_Out;
			VAR_Mask						:= HMI.Mask AND IN_MaskEn AND IN_AlarmEn ;
			VAR_Fault 						:= VAR_iFault;
		ELSE
			OUT_Scale[VAR_Index].ActValue 	:= HMI.PV[VAR_Index];
			VAR_Mask						:= HMI.Mask;
			VAR_Fault 						:= FALSE;
		END_IF

		IF VAR_Fault AND IN_AlarmEn THEN
			IF IN_FaultOutMode = CST_AI_FaultMode_Low THEN
				VAR_Out := IN_Scale[VAR_Index].ScaleLOW;
			ELSIF IN_FaultOutMode = CST_AI_FaultMode_High THEN
				VAR_Out := IN_Scale[VAR_Index].ScaleHIGH;
			END_IF
			OUT_Alarm := TRUE;
		ELSIF IN_Reset THEN
			OUT_Alarm := FALSE;
		END_IF

		IF IN_Scale[VAR_Index].HighLimitEn AND NOT VAR_Mask THEN
			TMR_TON_HighLimitDelay(	IN := (OUT_Scale[VAR_Index].ActValue >= IN_Scale[VAR_Index].HighLimitSP),
									PT := IN_Scale[VAR_Index].HighLimitDelay);

			IF TMR_TON_HighLimitDelay.Q THEN
				OUT_Scale[VAR_Index].HighLimit 	:= TRUE;
			ELSIF (OUT_Scale[VAR_Index].ActValue <= (IN_Scale[VAR_Index].HighLimitSP - IN_Scale[VAR_Index].HighLimitHyst)) THEN
				OUT_Scale[VAR_Index].HighLimit 	:= FALSE;
			END_IF
		ELSE
			OUT_Scale[VAR_Index].HighLimit := FALSE;
		END_IF

		IF IN_Scale[VAR_Index].LowLimitEn AND NOT VAR_Mask THEN
			TMR_TON_LowLimitDelay(	IN := (OUT_Scale[VAR_Index].ActValue <= IN_Scale[VAR_Index].LowLimitSP),
									PT := IN_Scale[VAR_Index].LowLimitDelay);

			IF TMR_TON_LowLimitDelay.Q THEN
				OUT_Scale[VAR_Index].LowLimit 	:= TRUE;
			ELSIF (OUT_Scale[VAR_Index].ActValue >= (IN_Scale[VAR_Index].LowLimitSP + IN_Scale[VAR_Index].LowLimitHyst)) THEN
				OUT_Scale[VAR_Index].LowLimit 	:= FALSE;
			END_IF
		ELSE
			OUT_Scale[VAR_Index].LowLimit := FALSE;
		END_IF

	(*****************************************************************)
	(*************************COMPARE MODE****************************)
	(*****************************************************************)
		IF VAR_Mask THEN
			VAR_SpReached := TRUE;
			VAR_Wait := FALSE;
		ELSE
			CASE IN_CompareMode OF
				CST_AI_Compare_OFF:
					VAR_SpReached		:= FALSE;
					VAR_Wait 			:= FALSE;
					HMI.SP[VAR_Index]	:= HMI.PV[VAR_Index];

				CST_AI_Compare_LT:
					VAR_SpReached 		:= OUT_Scale[VAR_Index].ActValue < (IN_Scale[VAR_Index].ActualSP + IN_Scale[VAR_Index].MinDev);
					VAR_Wait 			:= NOT VAR_SpReached;
					HMI.SP[VAR_Index]	:= IN_Scale[VAR_Index].ActualSP;

				CST_AI_Compare_GT:
					VAR_SpReached 		:= OUT_Scale[VAR_Index].ActValue > (IN_Scale[VAR_Index].ActualSP - IN_Scale[VAR_Index].MaxDev);
					VAR_Wait 			:= NOT VAR_SpReached;
					HMI.SP[VAR_Index]	:= IN_Scale[VAR_Index].ActualSP;

				CST_AI_Compare_EQ:
					VAR_SpReached 		:= (OUT_Scale[VAR_Index].ActValue < (IN_Scale[VAR_Index].ActualSP + IN_Scale[VAR_Index].MaxDev)) AND (OUT_Scale[VAR_Index].ActValue > (IN_Scale[VAR_Index].ActualSP - IN_Scale[VAR_Index].MinDev));
					VAR_Wait 			:= NOT VAR_SpReached;
					HMI.SP[VAR_Index]	:= IN_Scale[VAR_Index].ActualSP;

				CST_AI_Compare_ON:
					VAR_SpReached 		:= TRUE;
					VAR_Wait 			:= FALSE;
					HMI.SP[VAR_Index]	:= HMI.PV[VAR_Index];
			END_CASE
		END_IF
	ELSE
		OUT_SpReached 					:= TRUE;
		OUT_Scale[VAR_Index].LowLimit	:= FALSE;
		OUT_Scale[VAR_Index].HighLimit 	:= FALSE;
	END_IF

	TMR_TOF_SpReached(IN:= VAR_SpReached, PT:= IN_Scale[VAR_Index].WaitDelay);
	OUT_SpReached	:= TMR_TOF_SpReached.Q;

	(*****************************************************************)
	(***************************TOTALIZER*****************************)
	(*****************************************************************)
	IF IN_Scale[VAR_Index].HMITotEn THEN
		HMITotalizer(
			IN_Pulse			:= IO.DI_Pulse,
			IN_AnalogPV			:= VAR_Out,
			IN_PulseWeight		:= IN_Scale[VAR_Index].TotPulseWeight,
			IN_ConfigType		:= IN_Scale[VAR_Index].TotType,
			IN_Reset			:= IN_Scale[VAR_Index].HMITotReset OR HMI.ResetTot,
			OUT_TotalCounter	:= HMI.Tot[VAR_Index]);

		HMI.ConfigTot[VAR_Index]	:= TRUE;
	ELSE
		HMI.ConfigTot[VAR_Index]	:= FALSE;
		HMI.Tot[VAR_Index] 			:= 0.0;
	END_IF

	IF IN_PLCCounterEn THEN
		PLCCounter(
			IN_Pulse			:= IO.DI_Pulse,
			IN_AnalogPV			:= VAR_Out,
			IN_PulseWeight		:= IN_Scale[VAR_Index].TotPulseWeight,
			IN_ConfigType		:= IN_Scale[VAR_Index].TotType,
			IN_Reset			:= IN_Scale[VAR_Index].PLCCounterReset,
			OUT_TotalCounter	:= HMI.PV_Counter[VAR_Index]);

		HMI.ConfigCounter[VAR_Index]	:= TRUE;
	ELSE
		HMI.ConfigCounter[VAR_Index]	:= FALSE;
		HMI.PV_Counter[VAR_Index]		:= 0.0;
	END_IF

	OUT_Scale[VAR_Index].PLCCounterReached := (HMI.PV_Counter[VAR_Index] >= IN_Scale[VAR_Index].PLCCounterSP);

	HMI.ConfigAlarm					:= IN_AlarmEn;
	HMI.ConfigPresent 				:= IN_ConfigPresent;
	HMI.SP_Counter[VAR_Index]		:= IN_Scale[VAR_Index].PLCCounterSP;
	HMI.WaitCounter[VAR_Index]		:= IN_PLCCounterEn AND NOT OUT_Scale[VAR_Index].PLCCounterReached;
	HMI.Wait[VAR_Index]				:= VAR_Wait;
	HMI.Unit						:= VAR_Index;
	HMI.Alarm						:= OUT_Alarm;
	HMI.PV[VAR_Index]				:= OUT_Scale[VAR_Index].ActValue;

	IF NOT IN_Simulation THEN
		HMI.MaskEnable	:= IN_MaskEn;
		HMI.ConfigPopup	:= IN_ConfigPopup;
	ELSE
		HMI.MaskEnable	:= TRUE;
		HMI.ConfigPopup	:= TRUE;
	END_IF
END_FUNCTION_BLOCK

(* ---- Analog_In_Multiscale.st ---- *)
FUNCTION_BLOCK Analog_In_Multiscale
	IF IN_ConfigPresent THEN

	(*****************************************************************)
	(****************************VALUE SCALING************************)
	(*****************************************************************)
		IF IN_EngScale THEN
			VAR_ChannelActive := IO.AI_Raw < 32767;
		ELSE
			IF IN_0_20mA THEN
				VAR_ChannelActive := (IO.AI_Raw > 6000);
			ELSE
				VAR_ChannelActive := NOT ((IO.AI_Raw < -90) OR (IO.AI_Raw > 32767));
			END_IF
			OUT_RawOverflow 	:= (IO.AI_Raw > 32767) AND NOT HMI.Mask;
			OUT_RawUnderflow	:= NOT VAR_ChannelActive AND (IO.AI_Raw < 32767) AND NOT HMI.Mask;
		END_IF

		VAR_Index := IN_ScaleIndex;

		LCRLimScal_0_20mA(
			x	:= INT_TO_REAL(IO.AI_Raw),
			x1	:= 6553.4,
			y1	:= IN_Scale[VAR_Index].ScaleLOW,
			x2	:= 32767.0,
			y2	:= IN_Scale[VAR_Index].ScaleHIGH
			);

		LCRLimScal_4_20mA(
			x	:= INT_TO_REAL(IO.AI_Raw),
			x1	:= 0.0,
			y1	:= IN_Scale[VAR_Index].ScaleLOW,
			x2	:= 32767.0,
			y2	:= IN_Scale[VAR_Index].ScaleHIGH
			);

		IF VAR_ChannelActive THEN
			IF IN_EngScale THEN
				VAR_Out := INT_TO_REAL(IO.AI_Raw) / 10.0;
			ELSE
				IF IN_0_20mA THEN
					VAR_Out := LCRLimScal_0_20mA.y;
				ELSE
					VAR_Out := LCRLimScal_4_20mA.y;
				END_IF
			END_IF

			IF IN_Reset THEN
				VAR_iFault := FALSE;
			END_IF
		ELSE
			VAR_iFault := NOT VAR_Mask;
		END_IF

	(*****************************************************************)
	(***********************FAULTS AND LIMITS*************************)
	(*****************************************************************)
		IF NOT IN_Simulation THEN
			OUT_Scale[VAR_Index].ActValue 	:= VAR_Out;
			VAR_Mask						:= HMI.Mask AND IN_MaskEn AND IN_AlarmEn ;
			VAR_Fault 						:= VAR_iFault;
		ELSE
			OUT_Scale[VAR_Index].ActValue 	:= HMI.PV[VAR_Index];
			VAR_Mask						:= HMI.Mask;
			VAR_Fault 						:= FALSE;
		END_IF

		IF VAR_Fault AND IN_AlarmEn THEN
			IF IN_FaultOutMode = CST_AI_FaultMode_Low THEN
				VAR_Out := IN_Scale[VAR_Index].ScaleLOW;
			ELSIF IN_FaultOutMode = CST_AI_FaultMode_High THEN
				VAR_Out := IN_Scale[VAR_Index].ScaleHIGH;
			END_IF
			OUT_Alarm := TRUE;
		ELSIF IN_Reset THEN
			OUT_Alarm := FALSE;
		END_IF

		IF IN_Scale[VAR_Index].HighLimitEn AND NOT VAR_Mask THEN
			TMR_TON_HighLimitDelay(	IN := (OUT_Scale[VAR_Index].ActValue >= IN_Scale[VAR_Index].HighLimitSP),
									PT := IN_Scale[VAR_Index].HighLimitDelay);

			IF TMR_TON_HighLimitDelay.Q THEN
				OUT_Scale[VAR_Index].HighLimit 	:= TRUE;
			ELSIF (OUT_Scale[VAR_Index].ActValue <= (IN_Scale[VAR_Index].HighLimitSP - IN_Scale[VAR_Index].HighLimitHyst)) THEN
				OUT_Scale[VAR_Index].HighLimit 	:= FALSE;
			END_IF
		ELSE
			OUT_Scale[VAR_Index].HighLimit := FALSE;
		END_IF

		IF IN_Scale[VAR_Index].LowLimitEn AND NOT VAR_Mask THEN
			TMR_TON_LowLimitDelay(	IN := (OUT_Scale[VAR_Index].ActValue <= IN_Scale[VAR_Index].LowLimitSP),
									PT := IN_Scale[VAR_Index].LowLimitDelay);

			IF TMR_TON_LowLimitDelay.Q THEN
				OUT_Scale[VAR_Index].LowLimit 	:= TRUE;
			ELSIF (OUT_Scale[VAR_Index].ActValue >= (IN_Scale[VAR_Index].LowLimitSP + IN_Scale[VAR_Index].LowLimitHyst)) THEN
				OUT_Scale[VAR_Index].LowLimit 	:= FALSE;
			END_IF
		ELSE
			OUT_Scale[VAR_Index].LowLimit := FALSE;
		END_IF

	(*****************************************************************)
	(*************************COMPARE MODE****************************)
	(*****************************************************************)
		IF VAR_Mask THEN
			VAR_SpReached := TRUE;
			VAR_Wait := FALSE;
		ELSE
			CASE IN_CompareMode OF
				CST_AI_Compare_OFF:
					VAR_SpReached		:= FALSE;
					VAR_Wait 			:= FALSE;
					HMI.SP[VAR_Index]	:= HMI.PV[VAR_Index];

				CST_AI_Compare_LT:
					VAR_SpReached 		:= OUT_Scale[VAR_Index].ActValue < (IN_Scale[VAR_Index].ActualSP + IN_Scale[VAR_Index].MinDev);
					VAR_Wait 			:= NOT VAR_SpReached;
					HMI.SP[VAR_Index]	:= IN_Scale[VAR_Index].ActualSP;

				CST_AI_Compare_GT:
					VAR_SpReached 		:= OUT_Scale[VAR_Index].ActValue > (IN_Scale[VAR_Index].ActualSP - IN_Scale[VAR_Index].MaxDev);
					VAR_Wait 			:= NOT VAR_SpReached;
					HMI.SP[VAR_Index]	:= IN_Scale[VAR_Index].ActualSP;

				CST_AI_Compare_EQ:
					VAR_SpReached 		:= (OUT_Scale[VAR_Index].ActValue < (IN_Scale[VAR_Index].ActualSP + IN_Scale[VAR_Index].MaxDev)) AND (OUT_Scale[VAR_Index].ActValue > (IN_Scale[VAR_Index].ActualSP - IN_Scale[VAR_Index].MinDev));
					VAR_Wait 			:= NOT VAR_SpReached;
					HMI.SP[VAR_Index]	:= IN_Scale[VAR_Index].ActualSP;

				CST_AI_Compare_ON:
					VAR_SpReached 		:= TRUE;
					VAR_Wait 			:= FALSE;
					HMI.SP[VAR_Index]	:= HMI.PV[VAR_Index];
			END_CASE
		END_IF
	ELSE
		OUT_SpReached 					:= TRUE;
		OUT_Scale[VAR_Index].LowLimit	:= FALSE;
		OUT_Scale[VAR_Index].HighLimit 	:= FALSE;
	END_IF

	TMR_TOF_SpReached(IN:= VAR_SpReached, PT:= IN_Scale[VAR_Index].WaitDelay);
	OUT_SpReached	:= TMR_TOF_SpReached.Q;

	(*****************************************************************)
	(***************************TOTALIZER*****************************)
	(*****************************************************************)
	IF IN_Scale[VAR_Index].HMITotEn THEN
		HMITotalizer(
			IN_Pulse			:= IO.DI_Pulse,
			IN_AnalogPV			:= VAR_Out,
			IN_PulseWeight		:= IN_Scale[VAR_Index].TotPulseWeight,
			IN_ConfigType		:= IN_Scale[VAR_Index].TotType,
			IN_Reset			:= IN_Scale[VAR_Index].HMITotReset OR HMI.ResetTot,
			OUT_TotalCounter	:= HMI.Tot[VAR_Index]);

		HMI.ConfigTot[VAR_Index]	:= TRUE;
	ELSE
		HMI.ConfigTot[VAR_Index]	:= FALSE;
		HMI.Tot[VAR_Index] 			:= 0.0;
	END_IF

	IF IN_PLCCounterEn THEN
		PLCCounter(
			IN_Pulse			:= IO.DI_Pulse,
			IN_AnalogPV			:= VAR_Out,
			IN_PulseWeight		:= IN_Scale[VAR_Index].TotPulseWeight,
			IN_ConfigType		:= IN_Scale[VAR_Index].TotType,
			IN_Reset			:= IN_Scale[VAR_Index].PLCCounterReset,
			OUT_TotalCounter	:= HMI.PV_Counter[VAR_Index]);

		HMI.ConfigCounter[VAR_Index]	:= TRUE;
	ELSE
		HMI.ConfigCounter[VAR_Index]	:= FALSE;
		HMI.PV_Counter[VAR_Index]		:= 0.0;
	END_IF

	OUT_Scale[VAR_Index].PLCCounterReached := (HMI.PV_Counter[VAR_Index] >= IN_Scale[VAR_Index].PLCCounterSP);

	HMI.ConfigAlarm					:= IN_AlarmEn;
	HMI.ConfigPresent 				:= IN_ConfigPresent;
	HMI.SP_Counter[VAR_Index]		:= IN_Scale[VAR_Index].PLCCounterSP;
	HMI.WaitCounter[VAR_Index]		:= IN_PLCCounterEn AND NOT OUT_Scale[VAR_Index].PLCCounterReached;
	HMI.Wait[VAR_Index]				:= VAR_Wait;
	HMI.Unit						:= VAR_Index;
	HMI.Alarm						:= OUT_Alarm;
	HMI.PV[VAR_Index]				:= OUT_Scale[VAR_Index].ActValue;

	IF NOT IN_Simulation THEN
		HMI.MaskEnable	:= IN_MaskEn;
		HMI.ConfigPopup	:= IN_ConfigPopup;
	ELSE
		HMI.MaskEnable	:= TRUE;
		HMI.ConfigPopup	:= TRUE;
	END_IF
END_FUNCTION_BLOCK

(* ---- Digital_Obj.st ---- *)
FUNCTION_BLOCK Digital_Obj
	IF IN_ConfigPresent THEN
		VAR_Mask := IN_MaskEn AND HMI.Mask;
		IF VAR_Mask THEN
			VAR_Signal := IN_WaitOn AND NOT IN_WaitOff;
		ELSE
			VAR_Signal := IO.DI_Input;
		END_IF

		TMR_TON_SwOn(	IN := VAR_Signal,
						PT := IN_SwitchDelay);

		TMR_TON_SwOff(	IN := NOT VAR_Signal,
						PT := IN_SwitchDelay);

		IF TMR_TON_SwOn.Q THEN
			HMI.On := TRUE;
		ELSIF TMR_TON_SwOff.Q THEN
			HMI.On := FALSE;
		END_IF

		TMR_TON_OnAlarm(	IN := IN_Alarm AND IN_AlarmOnReq AND HMI.On AND NOT VAR_Mask,
							PT := IN_OnDelay);

		TMR_TON_OffAlarm(	IN := IN_Alarm AND IN_AlarmOffReq AND NOT HMI.On AND NOT VAR_Mask,
							PT := IN_OffDelay);

		IF (TMR_TON_OnAlarm.Q OR TMR_TON_OffAlarm.Q) THEN
			OUT_Alarm := TRUE;
		ELSIF IN_Reset THEN
			OUT_Alarm := FALSE ;
		END_IF

		TMR_TON_OnTime(	IN := HMI.On,
						PT := IN_OnDelay);

		TMR_TON_OffTime(IN := NOT HMI.On,
						PT := IN_OffDelay);

		OUT_OnDelayed	:= TMR_TON_OnTime.Q;
		OUT_OffDelayed	:= TMR_TON_OffTime.Q;

		OUT					:= HMI.On;
		HMI.ConfigPresent 	:= IN_ConfigPresent;
		HMI.ConfigAlarm 	:= IN_Alarm OR IN_MaskEn;
		HMI.Alarm 			:= OUT_Alarm;
		HMI.Wait			:= (IN_WaitOn AND NOT HMI.On) OR (IN_WaitOff AND HMI.On);
		HMI.MaskEnable		:= IN_MaskEn;
	ELSE
		OUT_Alarm			:= FALSE;
		OUT					:= FALSE;
		OUT_OffDelayed		:= FALSE;
		OUT_OnDelayed		:= FALSE;
		HMI.On 				:= FALSE;
		HMI.MaskEnable		:= FALSE;
		HMI.ConfigPresent 	:= FALSE;
		HMI.ConfigAlarm 	:= FALSE;
		HMI.Alarm 			:= FALSE;
		HMI.Wait			:= FALSE;
	END_IF
END_FUNCTION_BLOCK

FUNCTION_BLOCK GateDoorDigital_Obj
	IF IN_ConfigPresent THEN
		VAR_Signal := IO_Production.DI_Input;

		TMR_TON_ProdSwOn(	IN := VAR_Signal,
			PT := IN_SwitchDelay);

		TMR_TON_ProdSwOff(	IN := NOT VAR_Signal,
			PT := IN_SwitchDelay);

		IF TMR_TON_ProdSwOn.Q THEN
			HMI.Production.On := TRUE;
		ELSIF TMR_TON_ProdSwOff.Q THEN
			HMI.Production.On := FALSE;
		END_IF

		//Controllo se il sensore di Produzione è impegnato durante il CIP (AlarmOpenReq)
		TMR_TON_ProdOnAlarm(	IN := IN_Alarm AND IN_AlarmOpenReq AND HMI.Production.On AND NOT HMI.Production.Mask,
			PT := IN_OnDelay);

		//Controllo se il sensore di Produzione è disimpegnato durante la Produzione (AlarmCloseReq)
		TMR_TON_ProdOffAlarm(	IN := IN_Alarm AND IN_AlarmCloseReq AND NOT HMI.Production.On AND NOT HMI.Production.Mask,
			PT := IN_OffDelay);

		VAR_Signal := IN_SafetyClosed;

		TMR_TON_CleanSwOn(	IN := VAR_Signal,
			PT := IN_SwitchDelay);

		TMR_TON_CleanSwOff(	IN := NOT VAR_Signal,
			PT := IN_SwitchDelay);

		IF TMR_TON_CleanSwOn.Q THEN
			HMI.Cleaning.On := TRUE;
		ELSIF TMR_TON_CleanSwOff.Q THEN
			HMI.Cleaning.On := FALSE;
		END_IF

		//Controllo se il sensore di CIP è impegnato durante il Produzione (AlarmCloseReq)
		TMR_TON_CleanOnAlarm(	IN := IN_Alarm AND IN_AlarmCloseReq AND HMI.Cleaning.On AND NOT HMI.Cleaning.Mask,
			PT := IN_OnDelay);

		//Controllo se il sensore di CIP è impegnato durante il CIP (AlarmOpenReq)
		TMR_TON_CleanOffAlarm(	IN := IN_Alarm AND IN_AlarmOpenReq AND NOT HMI.Cleaning.On AND NOT HMI.Cleaning.Mask,
			PT := IN_OffDelay);

		VAR_ProdFault	:= (TMR_TON_ProdOnAlarm.Q OR TMR_TON_ProdOffAlarm.Q) OR (HMI.Production.On AND HMI.Cleaning.On);
		VAR_CleanFault	:= (TMR_TON_CleanOnAlarm.Q OR TMR_TON_CleanOffAlarm.Q) OR (HMI.Production.On AND HMI.Cleaning.On);

		IF VAR_ProdFault OR VAR_CleanFault THEN
			OUT_Alarm := TRUE;
		ELSIF IN_Reset THEN
			OUT_Alarm := FALSE ;
		END_IF

		OUT_Opened	:= HMI.Production.On AND NOT HMI.Cleaning.On;
		OUT_Closed	:= NOT HMI.Production.On AND HMI.Cleaning.On;

		HMI.Opened						:= OUT_Opened;
		HMI.ShortSafety					:= IN_SafetyShortCircuit;
		HMI.Production.ConfigPresent 	:= IN_ConfigPresent;
		HMI.Cleaning.ConfigPresent 		:= IN_ConfigPresent;
		HMI.Production.MaskEnable		:= FALSE;
		HMI.Cleaning.MaskEnable			:= FALSE;
		HMI.Production.ConfigAlarm 		:= IN_Alarm;
		HMI.Cleaning.ConfigAlarm 		:= IN_Alarm;
		HMI.Production.Alarm			:= VAR_ProdFault;
		HMI.Cleaning.Alarm				:= VAR_CleanFault;
		HMI.Production.Wait				:= (IN_WaitOpen AND NOT HMI.Production.On);
		HMI.Cleaning.Wait				:= (IN_WaitClose AND NOT HMI.Cleaning.On);
	ELSE
		OUT_Alarm						:= FALSE;
		OUT_Opened						:= IN_AlarmOpenReq;
		OUT_Closed						:= IN_AlarmCloseReq;
		HMI.Opened						:= TRUE;
		HMI.ShortSafety					:= FALSE;
		HMI.Production.On				:= TRUE;
		HMI.Cleaning.On					:= FALSE;
		HMI.Production.ConfigPresent 	:= FALSE;
		HMI.Cleaning.ConfigPresent 		:= FALSE;
		HMI.Production.MaskEnable		:= FALSE;
		HMI.Cleaning.MaskEnable			:= FALSE;
		HMI.Production.ConfigAlarm 		:= FALSE;
		HMI.Cleaning.ConfigAlarm 		:= FALSE;
		HMI.Production.Alarm			:= FALSE;
		HMI.Cleaning.Alarm				:= FALSE;
		HMI.Production.Wait				:= FALSE;
		HMI.Cleaning.Wait				:= FALSE;
	END_IF
END_FUNCTION_BLOCK

(* ---- Fan.st ---- *)
FUNCTION_BLOCK Fan_Obj
	IF NOT(IN_RoofType) THEN
		IF IN_ConfigPresent THEN
			VAR_ResetHMI := FALSE;

			VAR_AbsoluteFilter		:= FALSE;
			VAR_PreFilter			:= FALSE;
			VAR_PressurizedOnAlarm	:= FALSE;

			FOR VAR_i := 1 TO IN_FanNumber DO
				HMI.HMI_Pressurizer[VAR_i].ConfigPresent	:= TRUE;
				HMI.HMI_Pressurizer[VAR_i].ManEnable		:= TRUE;
				HMI.HMI_Pressurizer[VAR_i].MaskEnable		:= TRUE;

				VAR_Auto[VAR_i]	:= NOT HMI.HMI_Pressurizer[VAR_i].ManOff AND NOT HMI.HMI_Pressurizer[VAR_i].ManOn;

				IF NOT IN_Enable THEN
					VAR_OUT := 0;
				ELSIF VAR_Auto[VAR_i] THEN
					VAR_OUT := IN_AutoSpeed;
				ELSIF HMI.HMI_Pressurizer[VAR_i].ManOn THEN
					VAR_OUT := HMI.HMI_Pressurizer[VAR_i].OUT_Man;
				ELSE
					VAR_OUT := 0;
				END_IF

				IF IN_HMIAutoForce THEN
					HMI.HMI_Pressurizer[VAR_i].ManOff	:= FALSE;
					HMI.HMI_Pressurizer[VAR_i].ManOn	:= FALSE;
				END_IF

				VAR_OUT := LIMIT(0, VAR_OUT, 100);

				IO.Pressurizer[VAR_i].AO_Raw	:= REAL_TO_INT(VAR_OUT * 32767 /100);
				// LAMP

				IF IN_CgfHmiLampOn THEN
					HMI.HMI_Pressurizer[VAR_i].SS2P_Lamp.Enable := VAR_i = 1;//V4.A.A.1.7.0 to enable the first zone
					HMI.HMI_Pressurizer[VAR_i].SS2P_Lamp.Visibility := TRUE;
					HMI.HMI_Pressurizer[VAR_i].SS2P_Lamp.LampON := HMI.HMI_Pressurizer[1].SS2P_Lamp.ON;//V4.A.A.1.7.0 fan 1 is managing all the lamp on
					IO.Pressurizer[VAR_i].DO_Lighting := HMI.HMI_Pressurizer[VAR_i].SS2P_Lamp.LampON;
				ELSE
					HMI.HMI_Pressurizer[VAR_i].SS2P_Lamp.Enable := FALSE;
					HMI.HMI_Pressurizer[VAR_i].SS2P_Lamp.Visibility := FALSE;
					HMI.HMI_Pressurizer[VAR_i].SS2P_Lamp.ON	:= FALSE;
					IO.Pressurizer[VAR_i].DO_Lighting := FALSE;
				END_IF

				IF IN_Reset THEN
					ALARM.Pressurizer[VAR_i].AbsoluteFilterAlarm	:= FALSE;
					ALARM.Pressurizer[VAR_i].PrefilterAlarm			:= FALSE;
					ALARM.Pressurizer[VAR_i].PressurizedOnAlarm		:= FALSE;
					OUT_OverloadFault						:= FALSE;
				END_IF

				IF NOT IO.Pressurizer[VAR_i].DI_AbsoluteFilterAlarm AND NOT HMI.HMI_Pressurizer[VAR_i].Mask AND IN_Enable THEN
					ALARM.Pressurizer[VAR_i].AbsoluteFilterAlarm	:= TRUE;
				END_IF
				VAR_AbsoluteFilter	:= ALARM.Pressurizer[VAR_i].AbsoluteFilterAlarm OR VAR_AbsoluteFilter;

				IF NOT IO.Pressurizer[VAR_i].DI_PrefilterAlarm AND NOT HMI.HMI_Pressurizer[VAR_i].Mask AND IN_Enable THEN
					ALARM.Pressurizer[VAR_i].PrefilterAlarm	:= TRUE;
				END_IF
				VAR_PreFilter	:= ALARM.Pressurizer[VAR_i].PrefilterAlarm OR VAR_PreFilter;

				TMR_TON_OnDelay[VAR_i](	IN := VAR_OUT > 0,
										PT := T#10s);
				TMR_TON_OffDelay[VAR_i](IN := VAR_OUT = 0,
										PT := T#25s);

				IF ((TMR_TON_OnDelay[VAR_i].Q AND NOT IO.Pressurizer[VAR_i].DI_PressurizerON) OR
					(TMR_TON_OffDelay[VAR_i].Q AND IO.Pressurizer[VAR_i].DI_PressurizerON)) AND NOT HMI.HMI_Pressurizer[VAR_i].Mask AND IN_Enable THEN
					ALARM.Pressurizer[VAR_i].PressurizedOnAlarm := TRUE;
				END_IF
				VAR_PressurizedOnAlarm	:= ALARM.Pressurizer[VAR_i].PressurizedOnAlarm OR VAR_PressurizedOnAlarm;

				ALARM.PressurizerZone.AbsoluteFilterAlarm	:= VAR_AbsoluteFilter;
				ALARM.PressurizerZone.PrefilterAlarm		:= VAR_PreFilter;
				ALARM.PressurizerZone.PressurizedOnAlarm	:= VAR_PressurizedOnAlarm;

				HMI.HMI_Pressurizer[VAR_i].Alarm		:= OUT_OverloadFault OR ALARM.Pressurizer[VAR_i].PressurizedOnAlarm;
				HMI.HMI_Pressurizer[VAR_i].AlarmFilter	:= ALARM.Pressurizer[VAR_i].AbsoluteFilterAlarm OR ALARM.Pressurizer[VAR_i].PrefilterAlarm;
				HMI.HMI_Pressurizer[VAR_i].Out			:= (VAR_OUT > 0.0);
				HMI.HMI_Pressurizer[VAR_i].OUT_CV		:= VAR_OUT;
			END_FOR

			IF NOT IO.DI_OverloadOK THEN
				OUT_OverloadFault := TRUE;
			END_IF
			Out_Light	:= HMI.HMI_Pressurizer[1].SS2P_Lamp.LampON;// v4.A.A.1.7.0
			OUT_Alarm	:= OUT_OverloadFault OR VAR_AbsoluteFilter OR VAR_PreFilter OR VAR_PressurizedOnAlarm;
		ELSE
			IF NOT VAR_ResetHMI THEN
				FOR VAR_i := 1 TO 6 DO
					HMI.HMI_Pressurizer[VAR_i].Alarm			:= FALSE;
					HMI.HMI_Pressurizer[VAR_i].AlarmFilter		:= FALSE;
					HMI.HMI_Pressurizer[VAR_i].ConfigPresent	:= FALSE;
					HMI.HMI_Pressurizer[VAR_i].ManEnable		:= FALSE;
					HMI.HMI_Pressurizer[VAR_i].ManState			:= FALSE;
					HMI.HMI_Pressurizer[VAR_i].MaskEnable		:= FALSE;
					HMI.HMI_Pressurizer[VAR_i].Out				:= FALSE;
					HMI.HMI_Pressurizer[VAR_i].OUT_CV			:= 0.0;
				END_FOR
				VAR_ResetHMI := TRUE;
			END_IF
		Out_Light	:= FALSE;;// v4.A.A.1.7.0
		END_IF
	ELSE
		//Galvani ROOF
		IF IN_ConfigPresent THEN
			VAR_ResetHMI := FALSE;

			HMI.HMI_Galvani.ConfigPresent:= TRUE;
			HMI.HMI_Galvani.ManEnable		:= TRUE;
			HMI.HMI_Galvani.MaskEnable		:= TRUE;

			VAR_Auto_Gal	:= NOT HMI.HMI_Galvani.ManOff AND NOT HMI.HMI_Galvani.ManOn;

			IF NOT IN_Enable THEN
				VAR_GalvaniOn := FALSE;
			ELSIF VAR_Auto_Gal THEN
				VAR_GalvaniOn := TRUE;
				VAR_GalvaniFlowSet := IN_GalvaniRoofFlowSet;
			ELSIF HMI.HMI_Galvani.ManOn THEN
				VAR_GalvaniOn := TRUE;
				VAR_GalvaniFlowSet := HMI.HMI_Galvani.ManFlowSet;
			ELSE
				VAR_GalvaniOn := FALSE;
			END_IF

			IF IN_HMIAutoForce THEN
				HMI.HMI_Galvani.ManOff	:= FALSE;
				HMI.HMI_Galvani.ManOn	:= FALSE;
			END_IF

			// LAMP
			IF IN_CgfHmiLampOn THEN
				HMI.HMI_Galvani.SS2P_Lamp1.Enable := TRUE;
				HMI.HMI_Galvani.SS2P_Lamp1.Visibility := TRUE;
				HMI.HMI_Galvani.SS2P_Lamp1.LampON := HMI.HMI_Galvani.SS2P_Lamp1.ON;
				IO.GalvaniRoof.DO_LightingArea_1 := HMI.HMI_Galvani.SS2P_Lamp1.LampON;

				HMI.HMI_Galvani.SS2P_Lamp2.Enable := TRUE;
				HMI.HMI_Galvani.SS2P_Lamp2.Visibility := TRUE;
				HMI.HMI_Galvani.SS2P_Lamp2.LampON := HMI.HMI_Galvani.SS2P_Lamp2.ON;
				IO.GalvaniRoof.DO_LightingArea_2 := HMI.HMI_Galvani.SS2P_Lamp2.LampON;
			ELSE
				HMI.HMI_Galvani.SS2P_Lamp1.Enable := FALSE;
				HMI.HMI_Galvani.SS2P_Lamp1.Visibility := FALSE;
				HMI.HMI_Galvani.SS2P_Lamp1.ON	:= FALSE;
				IO.GalvaniRoof.DO_LightingArea_1 := FALSE;

				HMI.HMI_Galvani.SS2P_Lamp2.Enable := FALSE;
				HMI.HMI_Galvani.SS2P_Lamp2.Visibility := FALSE;
				HMI.HMI_Galvani.SS2P_Lamp2.ON	:= FALSE;
				IO.GalvaniRoof.DO_LightingArea_2 := FALSE;
			END_IF

			IF IN_Reset THEN
				ALARM.Galvani.AbsoluteFilterAlarm		:= FALSE;
				ALARM.Galvani.PrefilterExtAlarm			:= FALSE;
				ALARM.Galvani.PrefilterIntAlarm			:= FALSE;
				ALARM.Galvani.RunningAlarm				:= FALSE;
				ALARM.Galvani.CabinetAlarm	            := FALSE;
				OUT_OverloadFault						:= FALSE;
			END_IF

			IF NOT IO.GalvaniRoof.DI_AbsoluteFilterAlarm AND NOT HMI.HMI_Galvani.Mask AND IN_Enable THEN
				ALARM.Galvani.AbsoluteFilterAlarm	:= TRUE;
			END_IF

			IF NOT IO.GalvaniRoof.DI_PrefilterExtAlarm AND NOT HMI.HMI_Galvani.Mask AND IN_Enable THEN
				ALARM.Galvani.PrefilterExtAlarm	:= TRUE;
			END_IF

			IF NOT IO.GalvaniRoof.DI_PrefilterIntAlarm AND NOT HMI.HMI_Galvani.Mask AND IN_Enable THEN
				ALARM.Galvani.PrefilterIntAlarm	:= TRUE;
			END_IF

			IF NOT IO.GalvaniRoof.DI_CabinetPoweredOn AND NOT HMI.HMI_Galvani.Mask AND IN_Enable THEN
				ALARM.Galvani.CabinetAlarm	:= TRUE;
			END_IF

			TMR_TON_OnDelay_Gal(IN := VAR_GalvaniOn,
								PT := T#10s);

			TMR_TON_OffDelay_Gal(IN := NOT(VAR_GalvaniOn),
								PT := T#25s);

			IF ((TMR_TON_OnDelay_Gal.Q AND NOT IO.GalvaniRoof.DI_Running) OR
				(TMR_TON_OffDelay_Gal.Q AND IO.GalvaniRoof.DI_Running)) AND NOT HMI.HMI_Galvani.Mask AND IN_Enable THEN
				ALARM.Galvani.RunningAlarm := TRUE;
			END_IF

			IF NOT IO.DI_OverloadOK THEN
				OUT_OverloadFault := TRUE;
			END_IF

			IF NOT(VAR_Auto_Gal) THEN
				ALARM.Galvani.SysManSwitchedOff := NOT(VAR_GalvaniOn);
			END_IF

			IF VAR_Auto_Gal THEN
				ALARM.Galvani.SysSwitchedOff := NOT(VAR_GalvaniOn);
			END_IF

			HMI.HMI_Galvani.Alarm				:= ALARM.Galvani.RunningAlarm OR ALARM.Galvani.CabinetAlarm;
			HMI.HMI_Galvani.AlarmAbsoluteFilter	:= ALARM.Galvani.AbsoluteFilterAlarm;
			HMI.HMI_Galvani.AlarmPrefilterInt	:= ALARM.Galvani.PrefilterIntAlarm;
			HMI.HMI_Galvani.AlarmPrefilterExt	:= ALARM.Galvani.PrefilterExtAlarm;
			HMI.HMI_Galvani.Overload			:= OUT_OverloadFault;
			HMI.HMI_Galvani.Out					:= VAR_GalvaniOn;
			HMI.HMI_Galvani.FlowSet				:= VAR_GalvaniFlowSet;

			IO.GalvaniRoof.DO_Start := VAR_GalvaniOn;
			IO.GalvaniRoof.DO_FlowSet := VAR_GalvaniFlowSet;

			OUT_Alarm := 	ALARM.Galvani.RunningAlarm OR
							ALARM.Galvani.AbsoluteFilterAlarm OR
							ALARM.Galvani.PrefilterExtAlarm OR
							ALARM.Galvani.PrefilterIntAlarm OR
							OUT_OverloadFault OR
							ALARM.Galvani.CabinetAlarm;
		ELSE
			IF NOT VAR_ResetHMI THEN
				HMI.HMI_Galvani.Alarm					:= FALSE;
				HMI.HMI_Galvani.AlarmAbsoluteFilter		:= FALSE;
				HMI.HMI_Galvani.AlarmPrefilterExt		:= FALSE;
				HMI.HMI_Galvani.AlarmPrefilterInt		:= FALSE;
				HMI.HMI_Galvani.Overload				:= FALSE;
				HMI.HMI_Galvani.ConfigPresent			:= FALSE;
				HMI.HMI_Galvani.ManEnable				:= FALSE;
				HMI.HMI_Galvani.ManState				:= FALSE;
				HMI.HMI_Galvani.MaskEnable				:= FALSE;
				HMI.HMI_Galvani.Out						:= FALSE;
				VAR_ResetHMI := TRUE;
			END_IF
		END_IF
	END_IF
END_FUNCTION_BLOCK

(* ---- MotionFan_Obj.st ---- *)
FUNCTION_BLOCK MotionFan_Obj
	IF IN_ConfigPresent THEN
		(*****************************************************************)
		(*****************************START*******************************)
		IF VAR_Fault OR NOT IN_Enable THEN
			IO.DO_MotorON := FALSE;
		ELSE
			IO.DO_MotorON := IN_AutoCnd;
		END_IF

		(*****************************************************************)
		(**************************ALARM LOGIC****************************)
		(*****************************************************************)
		TMR_TON(IN := IO.DO_MotorON,
				PT := IN_FBKDelay);

		TMR_TOF(IN := NOT IO.DO_MotorON,
				PT := IN_FBKDelay);

		IF IN_Reset THEN
			VAR_ContactorFBK	:= FALSE;
			VAR_Isolated		:= FALSE;
			VAR_Overload		:= FALSE;
		END_IF

		IF ((TMR_TON.Q AND IO.DI_ContactorFBK) OR (TMR_TOF.Q AND NOT IO.DI_ContactorFBK)) THEN
			VAR_ContactorFBK := TRUE;
		END_IF

		IF NOT IO.DI_ManSwitchON THEN
			VAR_Isolated := TRUE;
		END_IF

		IF NOT IO.DI_OverloadOK THEN
			VAR_Overload := TRUE;
		END_IF

		VAR_Fault := (VAR_ContactorFBK OR VAR_Isolated OR VAR_Overload);

		(*****************************************************************)
		(******************************OUT********************************)
		(*****************************************************************)
		OUT_Running				:= IO.DO_MotorON;
		OUT_IsolatedFault		:= VAR_Isolated;
		OUT_ContactorFBKFault	:= VAR_ContactorFBK;
		OUT_OverloadFault		:= VAR_Overload;
		OUT_Alarm				:= VAR_Fault;
	ELSE
		OUT_Running				:= FALSE;
		OUT_IsolatedFault		:= FALSE;
		OUT_ContactorFBKFault	:= FALSE;
		OUT_OverloadFault		:= FALSE;
		OUT_Alarm				:= FALSE;
		IO.DO_MotorON			:= FALSE;
	END_IF
END_FUNCTION_BLOCK

(* ---- Motor_FC280_Vfd.st ---- *)
FUNCTION_BLOCK Motor_FC280_Vfd
	IF NOT VAR_FirstCycle THEN
		HMI_Motor.ManOff	:= FALSE;
		HMI_Motor.ManOn		:= FALSE;
		VAR_FirstCycle		:= TRUE;
	END_IF

	IF IN_ConfigPresent THEN
		(*****************************************************************)
		(**********************FREQUENCY AND START************************)
		(*****************************************************************)
		IF (EDGENEG(IN_ManEn) AND HMI_Motor.ManOn) OR IN_HMIAutoForce THEN
			HMI_Motor.ManOn	:= FALSE;
			HMI_Motor.ManOff	:= FALSE;
		END_IF

		VAR_Mask := HMI_Motor.Mask AND IN_MaskEn;
		VAR_Auto := NOT HMI_Motor.ManOff AND NOT HMI_Motor.ManOn;

		IF IN_JOGMode THEN
			VAR_AutoSpeed := 0.0;
			VAR_Start := IN_JOGCnd AND IN_Enable;
		ELSIF HMI_Motor.ManOn THEN
			VAR_AutoSpeed := HMI_Motor.OUT_Man;
			VAR_Start := IN_ManEn AND NOT IN_JOGMode AND IN_Enable;
		ELSIF VAR_Auto THEN
			VAR_AutoSpeed := IN_AutoSpeed;
			VAR_Start := IN_AutoCnd AND NOT IN_JOGMode AND IN_Enable;
		ELSE
			VAR_AutoSpeed := 0.0;
			VAR_Start := FALSE;
		END_IF

		VAR_AutoSpeed := LIMIT(IN_FrequencyMin, VAR_AutoSpeed, MIN(IN_FrequencyMax, IN_ScaleMax));

		IF NOT VAR_Start THEN
			VAR_AutoSpeed := 0.0;
		END_IF

		(*****************************************************************)
		(**************************START/STOP*****************************)
		(*****************************************************************)
		IF (NOT VAR_Isolated AND NOT VAR_RecSTW.Fault
			AND NOT VAR_Event.Over_Current AND NOT VAR_Event.Torque_Limit)
			AND	((IO_MotorFC280.DI_SafetyEnable AND VAR_RecSTW.T37_Ready) OR NOT IN_SafetyCtrlEn) THEN
			VAR_SendCTW.Start := VAR_Start;
		ELSE
			VAR_SendCTW.Start := FALSE;
		END_IF

		VAR_SendCTW.Reverse 				:= IN_Reverse;			//0- No function	1- Reverse
		VAR_SendCTW.Quick_Stop				:= NOT IN_QuickStopCmd;	//0- Quick Stop		1- Ramp
		VAR_SendCTW.Reset					:= IN_Reset;			//0- No function	1- Reset
		VAR_SendCTW.Coasting				:= NOT IN_CoastingCmd;	//0- Coasting		1- No Coasting
		VAR_SendCTW.DC_Brake				:= TRUE;				//0- DC Brake		1- Ramp
		VAR_SendCTW.Hold_Output_Frequency	:= TRUE;				//0- Hold Frequency	1- Ramp
		VAR_SendCTW.Data_Valid				:= TRUE;				//0- Data Invalid	1- Data Valid

		(*****************************************************************)
		(*****************************FAULT*******************************)
		(*****************************************************************)
		TMR_TON_RFeedBack(	IN := (VAR_SendCTW.Start AND VAR_AutoSpeed > 0) AND NOT OUT_InOperation AND NOT VAR_Mask,
							PT := IN_FBKDelay);

		TMR_TON_FaultFilter(	IN := VAR_RecSTW.Fault AND ((IO_MotorFC280.DI_SafetyEnable AND VAR_RecSTW.T37_Ready) OR NOT IN_SafetyCtrlEn),
								PT := T#200ms);

		TMR_TON_CurrentHigh(	IN := VAR_CurrentHigh,
								PT := T#5s);

		IF TMR_TON_FaultFilter.Q OR TMR_TON_CurrentHigh.Q OR TMR_TON_RFeedBack.Q OR
			VAR_Isolated OR VAR_Overload OR OUT_DriveSafetyFBKFault THEN
			VAR_Fault := TRUE;
		ELSIF IN_Reset THEN
			VAR_Fault := FALSE;
		END_IF

		OUT_DriveFault := VAR_Fault;

		IF (NOT IO_MotorFC280.DI_ManSwitchON OR (IN_FCD AND IO_MotorFC280.DI_OverloadOK AND NOT VAR_RecDI.T27 )) AND NOT VAR_Mask THEN //V4.A.A.1.6.13
			VAR_Isolated := TRUE;
		ELSIF IN_Reset THEN
			VAR_Isolated := FALSE;
		END_IF

		IF NOT IO_MotorFC280.DI_OverloadOK AND NOT VAR_Mask THEN
			VAR_Overload := TRUE;
		ELSIF IN_Reset THEN
			VAR_Overload := FALSE;
		END_IF

		TMR_TON_WarningFilter(	IN := (VAR_RecSTW.Warning AND NOT VAR_Mask) AND (IO_MotorFC280.DI_SafetyEnable OR NOT IN_SafetyCtrlEn),
								PT := T#1000ms);

		IF TMR_TON_WarningFilter.Q THEN
			OUT_Warning := TRUE;
		ELSIF IN_Reset THEN
			OUT_Warning := FALSE;
		END_IF

		(*****************************************************************)
		(********************SAFETY FEEDBACK FAULT************************)
		(*****************************************************************)
		TMR_TON_FBKTimeOut(	IN := ((VAR_RecSTW.T37_Ready XOR IO_MotorFC280.DI_SafetyEnable)) AND IN_SafetyCtrlEn,
							PT := T#3s);

		IF TMR_TON_FBKTimeOut.Q OR IO_MotorFC280.DI_SafetyFault THEN
			OUT_DriveSafetyFBKFault := TRUE;
		ELSIF IN_Reset THEN
			OUT_DriveSafetyFBKFault := FALSE;
		END_IF

		(*****************************************************************)
		(*************************ACTUAL SPEED****************************)
		(*****************************************************************)
		IO_DanfossFC280.Output.MRW := TRUNC((VAR_AutoSpeed / 100 )* 16384);

		IF IO_DanfossFC280.Input.MAV = 0 THEN
			OUT_ActualSpeed := 0;
		ELSE
			OUT_ActualSpeed := INT_TO_REAL(IO_DanfossFC280.Input.MAV)/ 16384 * 100;
		END_IF
		(*****************************************************************)
		(*****************************************************************)
		(*****************************************************************)

		IO_DanfossFC280.Output.CTW.2		:= VAR_SendCTW.DC_Brake;	(*not used*)
		IO_DanfossFC280.Output.CTW.3		:= VAR_SendCTW.Coasting;
		IO_DanfossFC280.Output.CTW.4		:= VAR_SendCTW.Quick_Stop;
		IO_DanfossFC280.Output.CTW.5		:= VAR_SendCTW.Hold_Output_Frequency; (*not used*)
		IO_DanfossFC280.Output.CTW.6		:= VAR_SendCTW.Start AND NOT IN_Simulation;
		IO_DanfossFC280.Output.CTW.7		:= VAR_SendCTW.Reset;
		IO_DanfossFC280.Output.CTW.8		:= VAR_SendCTW.Start AND IN_JOGMode;
		IO_DanfossFC280.Output.CTW.10		:= VAR_SendCTW.Data_Valid;
		IO_DanfossFC280.Output.CTW.15		:= VAR_SendCTW.Reverse;

		VAR_RecSTW.Fault 			:= IO_DanfossFC280.Input.STW.3;
		VAR_RecSTW.Warning 			:= IO_DanfossFC280.Input.STW.7;
		VAR_RecSTW.In_Operation 	:= IO_DanfossFC280.Input.STW.11;
//		VAR_RecSTW.T37_Ready 		:= IO_DanfossFC280.Input.STW.15;
		VAR_RecSTW.T37_Ready		:= IO_MotorFC280.DI_SafetyEnable; // da capire con danfoss
		//V4.A.A.1.6.13
		VAR_RecDI.T33				:= IO_DanfossFC280.Input.DigitalInput.0;
		VAR_RecDI.T32				:= IO_DanfossFC280.Input.DigitalInput.1;
		VAR_RecDI.T29				:= IO_DanfossFC280.Input.DigitalInput.2; //FCD:drive on safety
		VAR_RecDI.T27				:= IO_DanfossFC280.Input.DigitalInput.3; //FCD:status of the switch on board
		VAR_RecDI.T19				:= IO_DanfossFC280.Input.DigitalInput.4;
		VAR_RecDI.T18				:= IO_DanfossFC280.Input.DigitalInput.5;
//		VAR_RecDI.T37				:= IO_DanfossFC280.Input.DigitalInput.6; //FCD:safe stop

		OUT_ActualCurrent 		:= DINT_TO_REAL(IO_DanfossFC280.Input.ActCurrent) / 100;
		OUT_ActualFrequency		:= UDINT_TO_REAL(IO_DanfossFC280.Input.ActFreq) / 10;
		OUT_ActualPower 		:= DINT_TO_REAL(IO_DanfossFC280.Input.Power) /100;
		OUT_ActualTorque 		:= DINT_TO_REAL(IO_DanfossFC280.Input.Torque)/10;
		OUT_ActualSpeedRPM 		:= DINT_TO_REAL(IO_DanfossFC280.Input.SpeedRPM);
		OUT_SpeedReferece 	    := VAR_RecSTW.In_Operation AND IO_DanfossFC280.Output.CTW.7;
		OUT_InOperation 		:= VAR_RecSTW.In_Operation;
		OUT_IsolatedFault 		:= VAR_Isolated;
		OUT_OverloadFault 		:= VAR_Overload;

		(*****************************************************************)
		(****************************EVENT********************************)
		(*****************************************************************)

		(* Brake check 16#1*)
		VAR_Event.Brake_Check						:= IO_DanfossFC280.Input.ErrorCode.0;
		(* Power card over temperature 16#2 *)
		VAR_Event.Drive_Over_Temperature			:= IO_DanfossFC280.Input.ErrorCode.1;
		(* Earth fault 16#4 *)
		VAR_Event.Earth_Fault						:= IO_DanfossFC280.Input.ErrorCode.2;
		(* Control card over temperature 16#8 *)
		VAR_Event.Control_Card_Over_Temperature		:= IO_DanfossFC280.Input.ErrorCode.3;
		(* Control word timeout 16#10 *)
		VAR_Event.Controlword_timeout				:= IO_DanfossFC280.Input.ErrorCode.4;
		(* Over current 16#20 *)
		VAR_Event.Over_Current						:= IO_DanfossFC280.Input.ErrorCode.5;
		(* Torque limit 16#40 *)
		VAR_Event.Torque_Limit						:= IO_DanfossFC280.Input.ErrorCode.6;
		(* Motor thermistor over temp. 16#80 *)
		VAR_Event.Motor_Thermistor_Over_Temp		:= IO_DanfossFC280.Input.ErrorCode.7;
		(* Motor ETR over temperature 16#100 *)
		VAR_Event.Motor_ETR_Over_Temperature		:= IO_DanfossFC280.Input.ErrorCode.8;
		(* Inverter overloaded 16#200 *)
		VAR_Event.Inverter_Over_Loaded				:= IO_DanfossFC280.Input.ErrorCode.9;
		(* DC Link unver voltage 16#400 *)
		VAR_Event.DC_Link_Under_Voltage				:= IO_DanfossFC280.Input.ErrorCode.10;
		(* DC Link over voltage 16#800 *)
		VAR_Event.DC_Link_Over_Voltage				:= IO_DanfossFC280.Input.ErrorCode.11;
		(* Short circuit 16#1000 *)
		VAR_Event.Short_Circuit						:= IO_DanfossFC280.Input.ErrorCode.12;
		(* Inrush fault 16#2000 *)
		VAR_Event.Inrush_Fault						:= IO_DanfossFC280.Input.ErrorCode.13;
		(* Main phase loss 16#4000 *)
		VAR_Event.Mains_Phase_Loss					:= IO_DanfossFC280.Input.ErrorCode.14;
		(* AMA not ok 16#8000 *)
		VAR_Event.AMA_not_OK						:= IO_DanfossFC280.Input.ErrorCode.15;
		(* Live zero error 16# 10000 *)
		VAR_Event.Live_Zero_Error					:= IO_DanfossFC280.Input.ErrorCode.16;
		(* Internal Fault 16#20000 *)
		VAR_Event.Internal_Fault					:= IO_DanfossFC280.Input.ErrorCode.17;
		(* Brake overload 16#40000 *)
		VAR_Event.Brake_Resistor_Power_Limit		:= IO_DanfossFC280.Input.ErrorCode.18;
		(* Motor phase U is missing 16#80000 *)
		VAR_Event.Motor_Phase_U_Missing				:= IO_DanfossFC280.Input.ErrorCode.19;
		(* Motor phase V is missing 16#100000 *)
		VAR_Event.Motor_Phase_V_Missing				:= IO_DanfossFC280.Input.ErrorCode.20;
		(* Motor phase W is missing 16#200000 *)
		VAR_Event.Motor_Phase_W_Missing				:= IO_DanfossFC280.Input.ErrorCode.21;
		(* Fieldbus comm. fault 16#400000 *)
		VAR_Event.Fieldbus_Communication_Fault		:= IO_DanfossFC280.Input.ErrorCode.22;
		(* 24V supply fault 16#800000 *)
		VAR_Event._24V_Supply_Fault					:= IO_DanfossFC280.Input.ErrorCode.23;
		(* Mains failure 16#1000000 *)
		VAR_Event.Mains_Faliure						:= IO_DanfossFC280.Input.ErrorCode.24;
		(* 1.8V supply fault 16#2000000 *)
		VAR_Event._2V_Supply_Fault					:= IO_DanfossFC280.Input.ErrorCode.25;
		(* Brake resistor short circuit 16#4000000 *)
		VAR_Event.Brake_Resistor_Short_Circuit		:= IO_DanfossFC280.Input.ErrorCode.26;
		(* Brake chopper fault 16#8000000 *)
		VAR_Event.Brake_Chopper_Fault				:= IO_DanfossFC280.Input.ErrorCode.27;
		(* Option change 16#10000000 *)
		VAR_Event.Configuration_Option_Change		:= IO_DanfossFC280.Input.ErrorCode.28;
		(* Drive initialisation 16#20000000 *)
		VAR_Event.Drive_Initialisation				:= IO_DanfossFC280.Input.ErrorCode.29;
		(* Safe stop 16#40000000 *)
		VAR_Event.Safe_Stop							:= IO_DanfossFC280.Input.ErrorCode.30;
		(* Mechanical brake low 16#80000000 *)
		VAR_Event.Mecanical_Brake_Low				:= IO_DanfossFC280.Input.ErrorCode.31;

		VAR_CurrentHigh								:= IO_DanfossFC280.Input.STW_EX.7 ;

		(*****************************************************************)
		(******************************HMI********************************)
		(*****************************************************************)
		HMI_Motor.ConfigPresent	:= IN_ConfigPresent;
		HMI_Motor.Alarm			:= OUT_DriveFault;
		HMI_Motor.FeedBack		:= OUT_DriveSafetyFBKFault AND NOT VAR_Overload;
		HMI_Motor.Isolated		:= VAR_Isolated;
		HMI_Motor.Overload		:= VAR_Overload;
		HMI_Motor.Out			:= OUT_InOperation;
		HMI_Motor.MaskEnable	:= IN_MaskEn;
		HMI_Motor.ManEnable		:= IN_ManEn;
	   	HMI_Motor.OUT_CV		:= OUT_ActualFrequency;

		HMI_Danfoss.PCV.Alarm					:= (UDINT_TO_DINT (IO_DanfossFC280.Input.ErrorCode));
		HMI_Danfoss.PCD_Read.Frequency			:= OUT_ActualFrequency;
		HMI_Danfoss.PCD_Read.Main_Actual_Value	:= OUT_ActualSpeed;
		HMI_Danfoss.PCD_Read.Power				:= OUT_ActualPower;
		HMI_Danfoss.PCD_Read.Status_Word		:= IO_DanfossFC280.Input.STW;
		HMI_Danfoss.PCD_Read.Torque				:= OUT_ActualTorque;
		HMI_Danfoss.PCD_Read.Motor_Current		:= OUT_ActualCurrent;
		HMI_Danfoss.PCD_Read.Speed_RPM			:= OUT_ActualSpeedRPM;
	ELSE
		memset(ADR(HMI_Danfoss), 0, SIZEOF(HMI_Danfoss));
	END_IF
END_FUNCTION_BLOCK

(* ---- Motor_Std.st ---- *)
FUNCTION_BLOCK Motor_Std
	IF NOT VAR_FirstCycle THEN
		HMI.ManOff		:= FALSE;
		HMI.ManOn		:= FALSE;
		VAR_FirstCycle	:= TRUE;
	END_IF

	IF IN_ConfigPresent THEN
		(*****************************************************************)
		(*****************************START*******************************)
		(*****************************************************************)
		IF (EDGENEG(IN_ManEn) AND HMI.ManOn) OR IN_HMIAutoForce THEN
			HMI.ManOn	:= FALSE;
			HMI.ManOff	:= FALSE;
		END_IF

		VAR_Mask := HMI.Mask AND IN_MaskEn;
		VAR_Auto := NOT HMI.ManOff AND NOT HMI.ManOn;

		IF VAR_Fault OR NOT IN_Enable THEN
			IO.DO_MotorON := FALSE;
		ELSIF VAR_Auto THEN
			IO.DO_MotorON := IN_AutoCnd;
		ELSE
			IO.DO_MotorON := HMI.ManOn;
		END_IF

		(*****************************************************************)
		(**************************ALARM LOGIC****************************)
		(*****************************************************************)
		TMR_TON(IN := IO.DO_MotorON,
				PT := IN_FBKDelay);

		TMR_TOF(IN := NOT IO.DO_MotorON,
				PT := IN_FBKDelay);

		IF IN_Reset THEN
			VAR_ContactorFBK	:= FALSE;
			VAR_Isolated		:= FALSE;
			VAR_Overload		:= FALSE;
		END_IF

		IF ((TMR_TON.Q AND IO.DI_ContactorFBK) OR (TMR_TOF.Q AND NOT IO.DI_ContactorFBK)) AND NOT IN_ConfigType AND NOT VAR_Mask THEN
			VAR_ContactorFBK := NOT IN_Simulation;
		END_IF

		IO.DO_ShuntTrip := VAR_ContactorFBK;

		IF NOT IO.DI_ManSwitchON AND NOT VAR_Mask THEN
			VAR_Isolated := NOT IN_Simulation;
		END_IF

		IF NOT IO.DI_OverloadOK AND NOT IN_ConfigType AND NOT VAR_Mask THEN
			VAR_Overload := NOT IN_Simulation;
		END_IF

		VAR_Fault := (VAR_ContactorFBK OR VAR_Isolated OR VAR_Overload AND IN_Enable) AND NOT IN_Simulation;

		(*****************************************************************)
		(******************************HMI********************************)
		(*****************************************************************)
		HMI.Out				:= IO.DO_MotorON;
		HMI.Alarm			:= VAR_Fault;
		HMI.Isolated		:= VAR_Isolated;
		HMI.Overload		:= VAR_Overload;
		HMI.FeedBack		:= VAR_ContactorFBK;
		HMI.ConfigPresent	:= IN_ConfigPresent;
		HMI.ManEnable		:= IN_ManEn;
		HMI.MaskEnable		:= IN_MaskEn;

		(*****************************************************************)
		(******************************OUT********************************)
		(*****************************************************************)
		OUT_Running				:= IO.DO_MotorON;
		OUT_IsolatedFault		:= VAR_Isolated;
		OUT_ContactorFBKFault	:= VAR_ContactorFBK;
		OUT_OverloadFault		:= VAR_Overload;
		OUT_Alarm				:= VAR_Fault;
	ELSE
		memset(ADR(HMI), 0, SIZEOF(HMI));
		OUT_Running				:= FALSE;
		OUT_IsolatedFault		:= FALSE;
		OUT_ContactorFBKFault	:= FALSE;
		OUT_OverloadFault		:= FALSE;
		OUT_Alarm				:= FALSE;
		IO.DO_MotorON			:= FALSE;
	END_IF
END_FUNCTION_BLOCK

(* ---- Motor_Std_Fw_Bw.st ---- *)
FUNCTION_BLOCK Motor_Std_Fw_Bw
	IF NOT VAR_FirstCycle THEN
		HMI.ManOff		:= FALSE;
		HMI.ManOn		:= FALSE;
		VAR_FirstCycle	:= TRUE;
	END_IF

	IF IN_ConfigPresent THEN
		(*****************************************************************)
		(*****************************START*******************************)
		(*****************************************************************)
		IF (EDGENEG(IN_ManEn) AND HMI.ManOn) OR IN_HMIAutoForce THEN
			HMI.ManOn	:= FALSE;
			HMI.ManOff	:= FALSE;
		END_IF

		VAR_Mask := HMI.Mask AND IN_MaskEn;
		VAR_Auto := NOT HMI.ManOff AND NOT HMI.ManOn;

		IF VAR_Fault OR NOT IN_Enable THEN
			IO.DO_MotorFw := FALSE;
			IO.DO_MotorBw := FALSE;
		ELSIF VAR_Auto AND NOT IN_Backward THEN
			IO.DO_MotorFw := IN_AutoCnd;
			IO.DO_MotorBw := FALSE;
		ELSIF VAR_Auto AND IN_Backward THEN
			IO.DO_MotorFw := FALSE;
			IO.DO_MotorBw := IN_AutoCnd;
		ELSIF NOT VAR_Auto AND NOT IN_Backward	THEN
			IO.DO_MotorFw := HMI.ManOn;
		ELSIF NOT VAR_Auto AND IN_Backward	THEN
			IO.DO_MotorBw := HMI.ManOn;
		END_IF

		IF NOT IN_FbkCheck THEN
			IO.DI_ContactorFBK := NOT IO.DO_MotorFw AND NOT IO.DO_MotorBw;
		END_IF
		(*****************************************************************)
		(**************************ALARM LOGIC****************************)
		(*****************************************************************)
		TMR_TON(IN := IO.DO_MotorFw OR IO.DO_MotorBw ,
				PT := IN_FBKDelay);

		TMR_TOF(IN := NOT IO.DO_MotorFw AND NOT IO.DO_MotorBw,
				PT := IN_FBKDelay);

		IF IN_Reset THEN
			VAR_ContactorFBK	:= FALSE;
			VAR_Overload		:= FALSE;
			VAR_DiFault			:= FALSE;
		END_IF

		IF ((TMR_TON.Q AND IO.DI_ContactorFBK) OR (TMR_TOF.Q AND NOT IO.DI_ContactorFBK)) AND NOT IN_ConfigType AND NOT VAR_Mask THEN
			VAR_ContactorFBK := NOT IN_Simulation;
		END_IF

		IF IO.DI_Fault AND NOT VAR_Mask THEN
			VAR_DiFault := NOT IN_Simulation;
		END_IF

		IF NOT IO.DI_ManSwitchON AND NOT VAR_Mask THEN
			VAR_Isolated := NOT IN_Simulation;
		END_IF

		IF NOT IO.DI_OverloadOK AND NOT IN_ConfigType AND NOT VAR_Mask THEN
			VAR_Overload := NOT IN_Simulation;
		END_IF

		VAR_Fault := (VAR_ContactorFBK OR VAR_Isolated OR VAR_DiFault OR VAR_Overload AND IN_Enable) AND NOT IN_Simulation;

		(*****************************************************************)
		(******************************HMI********************************)
		(*****************************************************************)
		HMI.Out				:= IO.DO_MotorFw OR IO.DO_MotorBw;
		HMI.Alarm			:= VAR_Fault;
		HMI.Isolated		:= VAR_Isolated;
		HMI.Overload		:= VAR_Overload;
		HMI.FeedBack		:= VAR_ContactorFBK;
		HMI.ConfigPresent	:= IN_ConfigPresent;
		HMI.ManEnable		:= IN_ManEn;
		HMI.MaskEnable		:= IN_MaskEn;

		(*****************************************************************)
		(******************************OUT********************************)
		(*****************************************************************)
		OUT_Running				:= IO.DO_MotorFw OR IO.DO_MotorBw;
		OUT_IsolatedFault		:= VAR_Isolated;
		OUT_ContactorFBKFault	:= VAR_ContactorFBK;
		OUT_OverloadFault		:= VAR_Overload;
		OUT_Alarm				:= VAR_Fault;
	ELSE
		memset(ADR(HMI), 0, SIZEOF(HMI));
		OUT_Running				:= FALSE;
		OUT_ContactorFBKFault	:= FALSE;
		OUT_OverloadFault		:= FALSE;
		OUT_Alarm				:= FALSE;
		IO.DO_MotorFw 			:= FALSE;
		IO.DO_MotorBw           := FALSE;
	END_IF
END_FUNCTION_BLOCK

(* ---- Motor_Vfd.st ---- *)
FUNCTION_BLOCK Motor_Vfd
	IF NOT VAR_FirstCycle THEN
		HMI_Motor.ManOff	:= FALSE;
		HMI_Motor.ManOn		:= FALSE;
		VAR_FirstCycle		:= TRUE;
	END_IF

	IF IN_ConfigPresent THEN
		(*****************************************************************)
		(**********************FREQUENCY AND START************************)
		(*****************************************************************)
		IF (EDGENEG(IN_ManEn) AND HMI_Motor.ManOn) OR IN_HMIAutoForce THEN
			HMI_Motor.ManOn	:= FALSE;
			HMI_Motor.ManOff	:= FALSE;
		END_IF

		VAR_Mask := HMI_Motor.Mask AND IN_MaskEn;
		VAR_Auto := NOT HMI_Motor.ManOff AND NOT HMI_Motor.ManOn;

		IF IN_JOGMode THEN
			VAR_AutoSpeed := 0.0;
			VAR_Start := IN_JOGCnd AND IN_Enable;
		ELSIF HMI_Motor.ManOn THEN
			VAR_AutoSpeed := HMI_Motor.OUT_Man;
			VAR_Start := IN_ManEn AND NOT IN_JOGMode AND IN_Enable;
		ELSIF VAR_Auto THEN
			VAR_AutoSpeed := IN_AutoSpeed;
			VAR_Start := IN_AutoCnd AND NOT IN_JOGMode AND IN_Enable;
		ELSE
			VAR_AutoSpeed := 0.0;
			VAR_Start := FALSE;
		END_IF

		VAR_AutoSpeed := LIMIT(IN_FrequencyMin, VAR_AutoSpeed, MIN(IN_FrequencyMax, IN_ScaleMax));

		IF NOT VAR_Start THEN
			VAR_AutoSpeed := 0.0;
		END_IF

		(*****************************************************************)
		(**************************START/STOP*****************************)
		(*****************************************************************)
		IF (NOT VAR_Isolated AND NOT VAR_RecSTW.Fault
			AND NOT VAR_Event.Over_Current AND NOT VAR_Event.Torque_Limit)
			AND	((IO_Motor.DI_SafetyEnable AND VAR_RecSTW.T37_Ready) OR NOT IN_SafetyCtrlEn) THEN
			VAR_SendCTW.Start := VAR_Start;
		ELSE
			VAR_SendCTW.Start := FALSE;
		END_IF

		VAR_SendCTW.Reverse 				:= IN_Reverse;			//0- No function	1- Reverse
		VAR_SendCTW.Quick_Stop				:= NOT IN_QuickStopCmd;	//0- Quick Stop		1- Ramp
		VAR_SendCTW.Reset					:= IN_Reset;			//0- No function	1- Reset
		VAR_SendCTW.Coasting				:= NOT IN_CoastingCmd;	//0- Coasting		1- No Coasting
		VAR_SendCTW.DC_Brake				:= TRUE;				//0- DC Brake		1- Ramp
		VAR_SendCTW.Hold_Output_Frequency	:= TRUE;				//0- Hold Frequency	1- Ramp
		VAR_SendCTW.Data_Valid				:= TRUE;				//0- Data Invalid	1- Data Valid

		(*****************************************************************)
		(*****************************FAULT*******************************)
		(*****************************************************************)
		TMR_TON_RFeedBack(	IN := (VAR_SendCTW.Start AND VAR_AutoSpeed > 0) AND NOT OUT_InOperation AND NOT VAR_Mask,
							PT := IN_FBKDelay);

		TMR_TON_FaultFilter(	IN := VAR_RecSTW.Fault AND ((IO_Motor.DI_SafetyEnable AND VAR_RecSTW.T37_Ready) OR NOT IN_SafetyCtrlEn),
								PT := T#200ms);

		TMR_TON_CurrentHigh(	IN := VAR_CurrentHigh,
								PT := T#5s);

		IF TMR_TON_FaultFilter.Q OR TMR_TON_CurrentHigh.Q OR TMR_TON_RFeedBack.Q OR
			VAR_Isolated OR VAR_Overload OR OUT_DriveSafetyFBKFault THEN
			VAR_Fault := TRUE;
		ELSIF IN_Reset THEN
			VAR_Fault := FALSE;
		END_IF

		OUT_DriveFault := VAR_Fault;

		IF (NOT IO_Motor.DI_ManSwitchON OR (IN_FCD AND IO_Motor.DI_OverloadOK AND NOT VAR_RecDI.T27 )) AND NOT VAR_Mask THEN //V4.A.A.1.6.13
			VAR_Isolated := TRUE;
		ELSIF IN_Reset THEN
			VAR_Isolated := FALSE;
		END_IF

		IF NOT IO_Motor.DI_OverloadOK AND NOT VAR_Mask THEN
			VAR_Overload := TRUE;
		ELSIF IN_Reset THEN
			VAR_Overload := FALSE;
		END_IF

		TMR_TON_WarningFilter(	IN := (VAR_RecSTW.Warning AND NOT VAR_Mask) AND (IO_Motor.DI_SafetyEnable OR NOT IN_SafetyCtrlEn),
								PT := T#1000ms);

		IF TMR_TON_WarningFilter.Q THEN
			OUT_Warning := TRUE;
		ELSIF IN_Reset THEN
			OUT_Warning := FALSE;
		END_IF

		(*****************************************************************)
		(********************SAFETY FEEDBACK FAULT************************)
		(*****************************************************************)
		TMR_TON_FBKTimeOut(	IN := ((VAR_RecSTW.T37_Ready XOR IO_Motor.DI_SafetyEnable)) AND IN_SafetyCtrlEn,
							PT := T#3s);

		IF TMR_TON_FBKTimeOut.Q OR IO_Motor.DI_SafetyFault THEN
			OUT_DriveSafetyFBKFault := TRUE;
		ELSIF IN_Reset THEN
			OUT_DriveSafetyFBKFault := FALSE;
		END_IF

		(*****************************************************************)
		(*************************ACTUAL SPEED****************************)
		(*****************************************************************)
		IO_Danfoss.Output.MRW := TRUNC((VAR_AutoSpeed / 100 )* 16384);

		IF IO_Danfoss.Input.MAV = 0 THEN
			OUT_ActualSpeed := 0;
		ELSE
			OUT_ActualSpeed := INT_TO_REAL(IO_Danfoss.Input.MAV)/ 16384 * 100;
		END_IF
		(*****************************************************************)
		(*****************************************************************)
		(*****************************************************************)

		IO_Danfoss.Output.CTW.2		:= VAR_SendCTW.DC_Brake;	(*not used*)
		IO_Danfoss.Output.CTW.3		:= VAR_SendCTW.Coasting;
		IO_Danfoss.Output.CTW.4		:= VAR_SendCTW.Quick_Stop;
		IO_Danfoss.Output.CTW.5		:= VAR_SendCTW.Hold_Output_Frequency; (*not used*)
		IO_Danfoss.Output.CTW.6		:= VAR_SendCTW.Start AND NOT IN_Simulation;
		IO_Danfoss.Output.CTW.7		:= VAR_SendCTW.Reset;
		IO_Danfoss.Output.CTW.8		:= VAR_SendCTW.Start AND IN_JOGMode;
		IO_Danfoss.Output.CTW.10	:= VAR_SendCTW.Data_Valid;
		IO_Danfoss.Output.CTW.15	:= VAR_SendCTW.Reverse;

		VAR_RecSTW.Fault 			:= IO_Danfoss.Input.STW.3;
		VAR_RecSTW.Warning 			:= IO_Danfoss.Input.STW.7;
		VAR_RecSTW.In_Operation 	:= IO_Danfoss.Input.STW.11;
		VAR_RecSTW.T37_Ready 		:= IO_Danfoss.Input.STW.15;
		//V4.A.A.1.6.13
		VAR_RecDI.T33				:= IO_Danfoss.Input.DigitalInput.0;
		VAR_RecDI.T32				:= IO_Danfoss.Input.DigitalInput.1;
		VAR_RecDI.T29				:= IO_Danfoss.Input.DigitalInput.2; //FCD:drive on safety
		VAR_RecDI.T27				:= IO_Danfoss.Input.DigitalInput.3; //FCD:status of the switch on board
		VAR_RecDI.T19				:= IO_Danfoss.Input.DigitalInput.4;
		VAR_RecDI.T18				:= IO_Danfoss.Input.DigitalInput.5;
		VAR_RecDI.T37				:= IO_Danfoss.Input.DigitalInput.6; //FCD:safe stop

		OUT_ActualCurrent 		:= DINT_TO_REAL(IO_Danfoss.Input.ActCurrent) / 100;
		OUT_ActualFrequency		:= UINT_TO_REAL(IO_Danfoss.Input.ActFreq) / 10;
		OUT_ActualPower 		:= DINT_TO_REAL(IO_Danfoss.Input.Power) /100;
		OUT_ActualTorque 		:= DINT_TO_REAL(IO_Danfoss.Input.Torque)/10;
		OUT_ActualSpeedRPM 		:= DINT_TO_REAL(IO_Danfoss.Input.SpeedRPM);
		OUT_SpeedReferece 	    := VAR_RecSTW.In_Operation AND IO_Danfoss.Output.CTW.7;
		OUT_InOperation 		:= VAR_RecSTW.In_Operation;
		OUT_IsolatedFault 		:= VAR_Isolated;
		OUT_OverloadFault 		:= VAR_Overload;
		OUT_ActualDigitalState	:= VAR_RecDI;//v4.A.A.1.7.0
		(*****************************************************************)
		(****************************EVENT********************************)
		(*****************************************************************)

		(* Brake check 16#1*)
		VAR_Event.Brake_Check						:= IO_Danfoss.Input.ErrorCode.0;
		(* Power card over temperature 16#2 *)
		VAR_Event.Drive_Over_Temperature			:= IO_Danfoss.Input.ErrorCode.1;
		(* Earth fault 16#4 *)
		VAR_Event.Earth_Fault						:= IO_Danfoss.Input.ErrorCode.2;
		(* Control card over temperature 16#8 *)
		VAR_Event.Control_Card_Over_Temperature		:= IO_Danfoss.Input.ErrorCode.3;
		(* Control word timeout 16#10 *)
		VAR_Event.Controlword_timeout				:= IO_Danfoss.Input.ErrorCode.4;
		(* Over current 16#20 *)
		VAR_Event.Over_Current						:= IO_Danfoss.Input.ErrorCode.5;
		(* Torque limit 16#40 *)
		VAR_Event.Torque_Limit						:= IO_Danfoss.Input.ErrorCode.6;
		(* Motor thermistor over temp. 16#80 *)
		VAR_Event.Motor_Thermistor_Over_Temp		:= IO_Danfoss.Input.ErrorCode.7;
		(* Motor ETR over temperature 16#100 *)
		VAR_Event.Motor_ETR_Over_Temperature		:= IO_Danfoss.Input.ErrorCode.8;
		(* Inverter overloaded 16#200 *)
		VAR_Event.Inverter_Over_Loaded				:= IO_Danfoss.Input.ErrorCode.9;
		(* DC Link unver voltage 16#400 *)
		VAR_Event.DC_Link_Under_Voltage				:= IO_Danfoss.Input.ErrorCode.10;
		(* DC Link over voltage 16#800 *)
		VAR_Event.DC_Link_Over_Voltage				:= IO_Danfoss.Input.ErrorCode.11;
		(* Short circuit 16#1000 *)
		VAR_Event.Short_Circuit						:= IO_Danfoss.Input.ErrorCode.12;
		(* Inrush fault 16#2000 *)
		VAR_Event.Inrush_Fault						:= IO_Danfoss.Input.ErrorCode.13;
		(* Main phase loss 16#4000 *)
		VAR_Event.Mains_Phase_Loss					:= IO_Danfoss.Input.ErrorCode.14;
		(* AMA not ok 16#8000 *)
		VAR_Event.AMA_not_OK						:= IO_Danfoss.Input.ErrorCode.15;
		(* Live zero error 16# 10000 *)
		VAR_Event.Live_Zero_Error					:= IO_Danfoss.Input.ErrorCode.16;
		(* Internal Fault 16#20000 *)
		VAR_Event.Internal_Fault					:= IO_Danfoss.Input.ErrorCode.17;
		(* Brake overload 16#40000 *)
		VAR_Event.Brake_Resistor_Power_Limit		:= IO_Danfoss.Input.ErrorCode.18;
		(* Motor phase U is missing 16#80000 *)
		VAR_Event.Motor_Phase_U_Missing				:= IO_Danfoss.Input.ErrorCode.19;
		(* Motor phase V is missing 16#100000 *)
		VAR_Event.Motor_Phase_V_Missing				:= IO_Danfoss.Input.ErrorCode.20;
		(* Motor phase W is missing 16#200000 *)
		VAR_Event.Motor_Phase_W_Missing				:= IO_Danfoss.Input.ErrorCode.21;
		(* Fieldbus comm. fault 16#400000 *)
		VAR_Event.Fieldbus_Communication_Fault		:= IO_Danfoss.Input.ErrorCode.22;
		(* 24V supply fault 16#800000 *)
		VAR_Event._24V_Supply_Fault					:= IO_Danfoss.Input.ErrorCode.23;
		(* Mains failure 16#1000000 *)
		VAR_Event.Mains_Faliure						:= IO_Danfoss.Input.ErrorCode.24;
		(* 1.8V supply fault 16#2000000 *)
		VAR_Event._2V_Supply_Fault					:= IO_Danfoss.Input.ErrorCode.25;
		(* Brake resistor short circuit 16#4000000 *)
		VAR_Event.Brake_Resistor_Short_Circuit		:= IO_Danfoss.Input.ErrorCode.26;
		(* Brake chopper fault 16#8000000 *)
		VAR_Event.Brake_Chopper_Fault				:= IO_Danfoss.Input.ErrorCode.27;
		(* Option change 16#10000000 *)
		VAR_Event.Configuration_Option_Change		:= IO_Danfoss.Input.ErrorCode.28;
		(* Drive initialisation 16#20000000 *)
		VAR_Event.Drive_Initialisation				:= IO_Danfoss.Input.ErrorCode.29;
		(* Safe stop 16#40000000 *)
		VAR_Event.Safe_Stop							:= IO_Danfoss.Input.ErrorCode.30;
		(* Mechanical brake low 16#80000000 *)
		VAR_Event.Mecanical_Brake_Low				:= IO_Danfoss.Input.ErrorCode.31;

		VAR_CurrentHigh								:= IO_Danfoss.Input.STW_EX.7 ;

		(*****************************************************************)
		(******************************HMI********************************)
		(*****************************************************************)
		HMI_Motor.ConfigPresent	:= IN_ConfigPresent;
		HMI_Motor.Alarm			:= OUT_DriveFault;
		HMI_Motor.FeedBack		:= OUT_DriveSafetyFBKFault AND NOT VAR_Overload;
		HMI_Motor.Isolated		:= VAR_Isolated;
		HMI_Motor.Overload		:= VAR_Overload;
		HMI_Motor.Out			:= OUT_InOperation;
		HMI_Motor.MaskEnable	:= IN_MaskEn;
		HMI_Motor.ManEnable		:= IN_ManEn;
	   	HMI_Motor.OUT_CV		:= OUT_ActualFrequency;

		HMI_Danfoss.PCV.Alarm					:= (UDINT_TO_DINT (IO_Danfoss.Input.ErrorCode));
		HMI_Danfoss.PCD_Read.Frequency			:= OUT_ActualFrequency;
		HMI_Danfoss.PCD_Read.Main_Actual_Value	:= OUT_ActualSpeed;
		HMI_Danfoss.PCD_Read.Power				:= OUT_ActualPower;
		HMI_Danfoss.PCD_Read.Status_Word		:= IO_Danfoss.Input.STW;
		HMI_Danfoss.PCD_Read.Torque				:= OUT_ActualTorque;
		HMI_Danfoss.PCD_Read.Motor_Current		:= OUT_ActualCurrent;
		HMI_Danfoss.PCD_Read.Speed_RPM			:= OUT_ActualSpeedRPM;
	ELSE
		memset(ADR(HMI_Danfoss), 0, SIZEOF(HMI_Danfoss));
	END_IF
END_FUNCTION_BLOCK
